LIN {X 0,Y 481.428,Z 376.763,A -85,B 0,C 180,E1 -7015.184,E2 -7015.184} C_VEL
LIN {X 0,Y 481.4,Z 381.681,A -85,B 0,C 180,E1 -7016.232,E2 -7016.232} C_VEL
LIN {X 0,Y 481.223,Z 384.559,A -85,B 0,C 180,E1 -7017.069,E2 -7017.069} C_VEL
LIN {X 0,Y 480.948,Z 387.393,A -85,B 0,C 180,E1 -7018.324,E2 -7018.324} C_VEL
LIN {X 0,Y 480.921,Z 388.409,A -85,B 0,C 180,E1 -7019.162,E2 -7019.162} C_VEL
LIN {X 0,Y 480.91,Z 388.742,A -85,B 0,C 180,E1 -7019.999,E2 -7019.999} C_VEL
LIN {X 0,Y 480.91,Z 388.397,A -85,B 0,C 180,E1 -7020.836,E2 -7020.836} C_VEL
LIN {X 0,Y 480.929,Z 387.368,A -85,B 0,C 180,E1 -7021.674,E2 -7021.674} C_VEL
LIN {X 0,Y 481.008,Z 385.622,A -85,B 0,C 180,E1 -7022.511,E2 -7022.511} C_VEL
LIN {X 0,Y 481.16,Z 383.117,A -85,B 0,C 180,E1 -7023.348,E2 -7023.348} C_VEL
LIN {X 0,Y 481.355,Z 379.786,A -85,B 0,C 180,E1 -7024.185,E2 -7024.185} C_VEL
LIN {X 0,Y 481.453,Z 374.316,A -85,B 0,C 180,E1 -7025.233,E2 -7025.233} C_VEL
LIN {X 0,Y 481.518,Z 368.474,A -85,B 0,C 180,E1 -7026.073,E2 -7026.073} C_VEL
LIN {X 0,Y 481.67,Z 361.279,A -85,B 0,C 180,E1 -7026.891,E2 -7026.891} C_VEL
LIN {X 0,Y 481.799,Z 353.733,A -85,B 0,C 180,E1 -7027.543,E2 -7027.543} C_VEL
LIN {X 0,Y 482.018,Z 344.137,A -85,B 0,C 180,E1 -7028.172,E2 -7028.172} C_VEL
LIN {X 0,Y 481.92,Z 337.555,A -85,B 0,C 180,E1 -7028.49,E2 -7028.49} C_VEL
LIN {X 0,Y 481.191,Z 332.773,A -85,B 0,C 180,E1 -7028.714,E2 -7028.714} C_VEL
LIN {X 0,Y 481.282,Z 325.199,A -85,B 0,C 180,E1 -7031.935,E2 -7031.935} C_VEL
LIN {X 0,Y 481.289,Z 316.966,A -85,B 0,C 180,E1 -7035.471,E2 -7035.471} C_VEL
LIN {X 0,Y 481.36,Z 309.359,A -85,B 0,C 180,E1 -7038.735,E2 -7038.735} C_VEL
LIN {X 0,Y 481.373,Z 303.142,A -85,B 0,C 180,E1 -7041.406,E2 -7041.406} C_VEL
LIN {X 0,Y 481.425,Z 296.779,A -85,B 0,C 180,E1 -7044.125,E2 -7044.125} C_VEL
LIN {X 0,Y 481.494,Z 289.818,A -85,B 0,C 180,E1 -7047.08,E2 -7047.08} C_VEL
LIN {X 0,Y 481.611,Z 284.497,A -85,B 0,C 180,E1 -7049.327,E2 -7049.327} C_VEL
LIN {X 0,Y 481.644,Z 284.486,A -85,B 0,C 180,E1 -7052.675,E2 -7052.675} C_VEL
LIN {X 0,Y 481.624,Z 284.489,A -85,B 0,C 180,E1 -7055.709,E2 -7055.709} C_VEL
LIN {X 0,Y 481.659,Z 284.49,A -85,B 0,C 180,E1 -7058.858,E2 -7058.858} C_VEL
LIN {X 0,Y 481.632,Z 284.489,A -85,B 0,C 180,E1 -7062.16,E2 -7062.16} C_VEL
LIN {X 0,Y 481.647,Z 284.486,A -85,B 0,C 180,E1 -7065.541,E2 -7065.541} C_VEL
LIN {X 0,Y 481.648,Z 284.488,A -85,B 0,C 180,E1 -7068.957,E2 -7068.957} C_VEL
LIN {X 0,Y 481.648,Z 284.49,A -85,B 0,C 180,E1 -7071.991,E2 -7071.991} C_VEL
LIN {X 0,Y 481.684,Z 284.483,A -85,B 0,C 180,E1 -7075.317,E2 -7075.317} C_VEL
LIN {X 0,Y 481.639,Z 284.49,A -85,B 0,C 180,E1 -7078.311,E2 -7078.311} C_VEL
LIN {X 0,Y 481.697,Z 284.484,A -85,B 0,C 180,E1 -7081.218,E2 -7081.218} C_VEL
LIN {X 0,Y 481.696,Z 284.483,A -85,B 0,C 180,E1 -7084.042,E2 -7084.042} C_VEL
LIN {X 0,Y 481.641,Z 284.488,A -85,B 0,C 180,E1 -7087.14,E2 -7087.14} C_VEL
LIN {X 0,Y 480.959,Z 284.576,A -85,B 0,C 180,E1 -7087.838,E2 -7087.838} C_VEL
LIN {X 0,Y 478.104,Z 284.933,A -85,B 0,C 180,E1 -7088.971,E2 -7088.971} C_VEL
LIN {X 0,Y 475.715,Z 285.227,A -85,B 0,C 180,E1 -7089.885,E2 -7089.885} C_VEL
LIN {X 0,Y 474.713,Z 285.353,A -85,B 0,C 180,E1 -7090.591,E2 -7090.591} C_VEL
LIN {X 0,Y 474.644,Z 285.362,A -85,B 0,C 180,E1 -7090.83,E2 -7090.83} C_VEL
LIN {X 0,Y 474.668,Z 285.357,A -85,B 0,C 180,E1 -7094.232,E2 -7094.232} C_VEL
LIN {X 0,Y 474.688,Z 285.353,A -85,B 0,C 180,E1 -7097.724,E2 -7097.724} C_VEL
LIN {X 0,Y 474.688,Z 285.357,A -85,B 0,C 180,E1 -7100.627,E2 -7100.627} C_VEL
LIN {X 0,Y 474.687,Z 285.353,A -85,B 0,C 180,E1 -7103.198,E2 -7103.198} C_VEL
LIN {X 0,Y 474.73,Z 285.348,A -85,B 0,C 180,E1 -7104.904,E2 -7104.904} C_VEL
LIN {X 0,Y 474.861,Z 285.331,A -85,B 0,C 180,E1 -7107.455,E2 -7107.455} C_VEL
LIN {X 0,Y 474.866,Z 285.337,A -85,B 0,C 180,E1 -7110,E2 -7110} C_VEL
LIN {X 0,Y 474.862,Z 285.331,A -85,B 0,C 180,E1 -7112.545,E2 -7112.545} C_VEL
LIN {X 0,Y 474.742,Z 285.35,A -85,B 0,C 180,E1 -7115.948,E2 -7115.948} C_VEL
LIN {X 0,Y 474.699,Z 285.352,A -85,B 0,C 180,E1 -7118.514,E2 -7118.514} C_VEL
LIN {X 0,Y 474.691,Z 285.354,A -85,B 0,C 180,E1 -7121.963,E2 -7121.963} C_VEL
LIN {X 0,Y 474.688,Z 285.357,A -85,B 0,C 180,E1 -7125.456,E2 -7125.456} C_VEL
LIN {X 0,Y 474.654,Z 285.362,A -85,B 0,C 180,E1 -7129.011,E2 -7129.011} C_VEL
LIN {X 0,Y 474.579,Z 285.368,A -85,B 0,C 180,E1 -7131.729,E2 -7131.729} C_VEL
LIN {X 0,Y 474.649,Z 285.362,A -85,B 0,C 180,E1 -7134.494,E2 -7134.494} C_VEL
LIN {X 0,Y 474.688,Z 285.354,A -85,B 0,C 180,E1 -7137.339,E2 -7137.339} C_VEL
LIN {X 0,Y 474.601,Z 285.366,A -85,B 0,C 180,E1 -7140.812,E2 -7140.812} C_VEL
LIN {X 0,Y 474.629,Z 285.365,A -85,B 0,C 180,E1 -7143.985,E2 -7143.985} C_VEL
LIN {X 0,Y 474.566,Z 285.369,A -85,B 0,C 180,E1 -7146.901,E2 -7146.901} C_VEL
LIN {X 0,Y 474.619,Z 285.366,A -85,B 0,C 180,E1 -7149.649,E2 -7149.649} C_VEL
LIN {X 0,Y 474.606,Z 285.365,A -85,B 0,C 180,E1 -7152.935,E2 -7152.935} C_VEL
LIN {X 0,Y 474.595,Z 285.366,A -85,B 0,C 180,E1 -7155.896,E2 -7155.896} C_VEL
LIN {X 0,Y 474.6,Z 285.37,A -85,B 0,C 180,E1 -7159.045,E2 -7159.045} C_VEL
LIN {X 0,Y 474.599,Z 285.364,A -85,B 0,C 180,E1 -7161.706,E2 -7161.706} C_VEL
LIN {X 0,Y 474.611,Z 285.368,A -85,B 0,C 180,E1 -7164.726,E2 -7164.726} C_VEL
LIN {X 0,Y 474.621,Z 285.36,A -85,B 0,C 180,E1 -7167.788,E2 -7167.788} C_VEL
LIN {X 0,Y 474.702,Z 285.409,A -85,B 0,C 180,E1 -7169.68,E2 -7169.68} C_VEL
LIN {X 0,Y 474.647,Z 289.554,A -85,B 0,C 180,E1 -7171.719,E2 -7171.719} C_VEL
LIN {X 0,Y 474.489,Z 295.509,A -85,B 0,C 180,E1 -7174.625,E2 -7174.625} C_VEL
LIN {X 0,Y 474.341,Z 301.144,A -85,B 0,C 180,E1 -7177.344,E2 -7177.344} C_VEL
LIN {X 0,Y 474.256,Z 306.861,A -85,B 0,C 180,E1 -7180.074,E2 -7180.074} C_VEL
LIN {X 0,Y 474.132,Z 312.578,A -85,B 0,C 180,E1 -7182.756,E2 -7182.756} C_VEL
LIN {X 0,Y 474.044,Z 318.251,A -85,B 0,C 180,E1 -7185.403,E2 -7185.403} C_VEL
LIN {X 0,Y 474.062,Z 324.061,A -85,B 0,C 180,E1 -7188.086,E2 -7188.086} C_VEL
LIN {X 0,Y 473.949,Z 330.434,A -85,B 0,C 180,E1 -7190.963,E2 -7190.963} C_VEL
LIN {X 0,Y 475.276,Z 340.728,A -85,B 0,C 180,E1 -7191.444,E2 -7191.444} C_VEL
LIN {X 0,Y 475.007,Z 350.2,A -85,B 0,C 180,E1 -7192.028,E2 -7192.028} C_VEL
LIN {X 0,Y 474.815,Z 358.727,A -85,B 0,C 180,E1 -7192.731,E2 -7192.731} C_VEL
LIN {X 0,Y 474.55,Z 367.023,A -85,B 0,C 180,E1 -7193.624,E2 -7193.624} C_VEL
LIN {X 0,Y 474.497,Z 373.154,A -85,B 0,C 180,E1 -7194.476,E2 -7194.476} C_VEL
LIN {X 0,Y 474.346,Z 379.082,A -85,B 0,C 180,E1 -7195.54,E2 -7195.54} C_VEL
LIN {X 0,Y 474.117,Z 383.478,A -85,B 0,C 180,E1 -7196.602,E2 -7196.602} C_VEL
LIN {X 0,Y 473.955,Z 386.076,A -85,B 0,C 180,E1 -7197.451,E2 -7197.451} C_VEL
LIN {X 0,Y 473.87,Z 387.921,A -85,B 0,C 180,E1 -7198.301,E2 -7198.301} C_VEL
LIN {X 0,Y 473.857,Z 389.063,A -85,B 0,C 180,E1 -7199.151,E2 -7199.151} C_VEL
LIN {X 0,Y 473.861,Z 389.533,A -85,B 0,C 180,E1 -7200.001,E2 -7200.001} C_VEL
LIN {X 0,Y 473.873,Z 389.335,A -85,B 0,C 180,E1 -7200.851,E2 -7200.851} C_VEL
LIN {X 0,Y 473.906,Z 388.472,A -85,B 0,C 180,E1 -7201.701,E2 -7201.701} C_VEL
LIN {X 0,Y 473.99,Z 386.922,A -85,B 0,C 180,E1 -7202.551,E2 -7202.551} C_VEL
LIN {X 0,Y 474.162,Z 384.636,A -85,B 0,C 180,E1 -7203.4,E2 -7203.4} C_VEL
LIN {X 0,Y 474.331,Z 381.561,A -85,B 0,C 180,E1 -7204.25,E2 -7204.25} C_VEL
LIN {X 0,Y 474.604,Z 376.463,A -85,B 0,C 180,E1 -7205.311,E2 -7205.311} C_VEL
LIN {X 0,Y 474.665,Z 371.191,A -85,B 0,C 180,E1 -7206.163,E2 -7206.163} C_VEL
LIN {X 0,Y 474.887,Z 364.006,A -85,B 0,C 180,E1 -7207.07,E2 -7207.07} C_VEL
LIN {X 0,Y 475.278,Z 354.988,A -85,B 0,C 180,E1 -7207.937,E2 -7207.937} C_VEL
LIN {X 0,Y 475.511,Z 345.724,A -85,B 0,C 180,E1 -7208.607,E2 -7208.607} C_VEL
LIN {X 0,Y 475.411,Z 339.085,A -85,B 0,C 180,E1 -7208.984,E2 -7208.984} C_VEL
LIN {X 0,Y 474.159,Z 332.143,A -85,B 0,C 180,E1 -7209.331,E2 -7209.331} C_VEL
LIN {X 0,Y 474.254,Z 326.504,A -85,B 0,C 180,E1 -7212.024,E2 -7212.024} C_VEL
LIN {X 0,Y 474.432,Z 319.008,A -85,B 0,C 180,E1 -7215.66,E2 -7215.66} C_VEL
LIN {X 0,Y 474.594,Z 312.239,A -85,B 0,C 180,E1 -7219.014,E2 -7219.014} C_VEL
LIN {X 0,Y 474.769,Z 306.861,A -85,B 0,C 180,E1 -7221.721,E2 -7221.721} C_VEL
LIN {X 0,Y 474.976,Z 301.509,A -85,B 0,C 180,E1 -7224.476,E2 -7224.476} C_VEL
LIN {X 0,Y 475.239,Z 295.854,A -85,B 0,C 180,E1 -7227.463,E2 -7227.463} C_VEL
LIN {X 0,Y 475.353,Z 290.917,A -85,B 0,C 180,E1 -7230.179,E2 -7230.179} C_VEL
LIN {X 0,Y 474.938,Z 286.999,A -85,B 0,C 180,E1 -7232.491,E2 -7232.491} C_VEL
LIN {X 0,Y 474.677,Z 285.361,A -85,B 0,C 180,E1 -7233.594,E2 -7233.594} C_VEL
LIN {X 0,Y 474.594,Z 285.37,A -85,B 0,C 180,E1 -7236.324,E2 -7236.324} C_VEL
LIN {X 0,Y 474.633,Z 285.365,A -85,B 0,C 180,E1 -7239.648,E2 -7239.648} C_VEL
LIN {X 0,Y 474.62,Z 285.367,A -85,B 0,C 180,E1 -7242.935,E2 -7242.935} C_VEL
LIN {X 0,Y 474.611,Z 285.367,A -85,B 0,C 180,E1 -7245.895,E2 -7245.895} C_VEL
LIN {X 0,Y 474.633,Z 285.366,A -85,B 0,C 180,E1 -7249.041,E2 -7249.041} C_VEL
LIN {X 0,Y 474.615,Z 285.368,A -85,B 0,C 180,E1 -7251.704,E2 -7251.704} C_VEL
LIN {X 0,Y 474.671,Z 285.497,A -85,B 0,C 180,E1 -7254.989,E2 -7254.989} C_VEL
LIN {X 0,Y 476.098,Z 291.334,A -85,B 0,C 180,E1 -7257.291,E2 -7257.291} C_VEL
LIN {X 0,Y 477.894,Z 299.615,A -85,B 0,C 180,E1 -7259.999,E2 -7259.999} C_VEL
LIN {X 0,Y 478.476,Z 303.1,A -85,B 0,C 180,E1 -7261.006,E2 -7261.006} C_VEL
LIN {X 0,Y 478.091,Z 308.638,A -85,B 0,C 180,E1 -7262.415,E2 -7262.415} C_VEL
LIN {X 0,Y 476.789,Z 322.51,A -85,B 0,C 180,E1 -7265.624,E2 -7265.624} C_VEL
LIN {X 0,Y 475.729,Z 339.255,A -85,B 0,C 180,E1 -7269.234,E2 -7269.234} C_VEL
LIN {X 0,Y 475.019,Z 355.708,A -85,B 0,C 180,E1 -7272.566,E2 -7272.566} C_VEL
LIN {X 0,Y 474.627,Z 369.075,A -85,B 0,C 180,E1 -7275.174,E2 -7275.174} C_VEL
LIN {X 0,Y 476.028,Z 383.097,A -85,B 0,C 180,E1 -7275.546,E2 -7275.546} C_VEL
LIN {X 0,Y 476.321,Z 388.808,A -85,B 0,C 180,E1 -7275.746,E2 -7275.746} C_VEL
LIN {X 0,Y 475.977,Z 401.249,A -85,B 0,C 180,E1 -7276.28,E2 -7276.28} C_VEL
LIN {X 0,Y 475.522,Z 413.187,A -85,B 0,C 180,E1 -7276.974,E2 -7276.974} C_VEL
LIN {X 0,Y 475.283,Z 423.595,A -85,B 0,C 180,E1 -7277.746,E2 -7277.746} C_VEL
LIN {X 0,Y 474.806,Z 433.942,A -85,B 0,C 180,E1 -7278.69,E2 -7278.69} C_VEL
LIN {X 0,Y 474.46,Z 443.425,A -85,B 0,C 180,E1 -7279.761,E2 -7279.761} C_VEL
LIN {X 0,Y 474.221,Z 452.603,A -85,B 0,C 180,E1 -7281.048,E2 -7281.048} C_VEL
LIN {X 0,Y 474.043,Z 459.976,A -85,B 0,C 180,E1 -7282.332,E2 -7282.332} C_VEL
LIN {X 0,Y 473.877,Z 466.576,A -85,B 0,C 180,E1 -7283.809,E2 -7283.809} C_VEL
LIN {X 0,Y 473.852,Z 470.404,A -85,B 0,C 180,E1 -7284.894,E2 -7284.894} C_VEL
LIN {X 0,Y 473.898,Z 472.829,A -85,B 0,C 180,E1 -7285.748,E2 -7285.748} C_VEL
LIN {X 0,Y 473.92,Z 474.806,A -85,B 0,C 180,E1 -7286.599,E2 -7286.599} C_VEL
LIN {X 0,Y 473.883,Z 476.298,A -85,B 0,C 180,E1 -7287.45,E2 -7287.45} C_VEL
LIN {X 0,Y 473.758,Z 478.001,A -85,B 0,C 180,E1 -7289.15,E2 -7289.15} C_VEL
LIN {X 0,Y 473.761,Z 478.249,A -85,B 0,C 180,E1 -7290,E2 -7290} C_VEL
LIN {X 0,Y 473.754,Z 478.042,A -85,B 0,C 180,E1 -7290.85,E2 -7290.85} C_VEL
LIN {X 0,Y 473.881,Z 476.432,A -85,B 0,C 180,E1 -7292.55,E2 -7292.55} C_VEL
LIN {X 0,Y 473.904,Z 474.976,A -85,B 0,C 180,E1 -7293.401,E2 -7293.401} C_VEL
LIN {X 0,Y 473.81,Z 471.936,A -85,B 0,C 180,E1 -7294.679,E2 -7294.679} C_VEL
LIN {X 0,Y 473.905,Z 467.814,A -85,B 0,C 180,E1 -7295.959,E2 -7295.959} C_VEL
LIN {X 0,Y 474.017,Z 461.448,A -85,B 0,C 180,E1 -7297.454,E2 -7297.454} C_VEL
LIN {X 0,Y 474.181,Z 454.486,A -85,B 0,C 180,E1 -7298.738,E2 -7298.738} C_VEL
LIN {X 0,Y 474.428,Z 445.714,A -85,B 0,C 180,E1 -7300.024,E2 -7300.024} C_VEL
LIN {X 0,Y 474.835,Z 435.719,A -85,B 0,C 180,E1 -7301.202,E2 -7301.202} C_VEL
LIN {X 0,Y 475.243,Z 426.23,A -85,B 0,C 180,E1 -7302.105,E2 -7302.105} C_VEL
LIN {X 0,Y 475.538,Z 415.711,A -85,B 0,C 180,E1 -7302.917,E2 -7302.917} C_VEL
LIN {X 0,Y 475.936,Z 403.316,A -85,B 0,C 180,E1 -7303.666,E2 -7303.666} C_VEL
LIN {X 0,Y 476.298,Z 391.532,A -85,B 0,C 180,E1 -7304.2,E2 -7304.2} C_VEL
LIN {X 0,Y 476.195,Z 383.965,A -85,B 0,C 180,E1 -7304.462,E2 -7304.462} C_VEL
LIN {X 0,Y 474.685,Z 369.599,A -85,B 0,C 180,E1 -7304.852,E2 -7304.852} C_VEL
LIN {X 0,Y 475.239,Z 353.202,A -85,B 0,C 180,E1 -7308.093,E2 -7308.093} C_VEL
LIN {X 0,Y 476.031,Z 335.475,A -85,B 0,C 180,E1 -7311.66,E2 -7311.66} C_VEL
LIN {X 0,Y 476.93,Z 318.979,A -85,B 0,C 180,E1 -7315.066,E2 -7315.066} C_VEL
LIN {X 0,Y 477.984,Z 303.66,A -85,B 0,C 180,E1 -7318.306,E2 -7318.306} C_VEL
LIN {X 0,Y 477.87,Z 300.392,A -85,B 0,C 180,E1 -7319.034,E2 -7319.034} C_VEL
LIN {X 0,Y 475.231,Z 288.352,A -85,B 0,C 180,E1 -7321.917,E2 -7321.917} C_VEL
LIN {X 0,Y 474.647,Z 285.363,A -85,B 0,C 180,E1 -7322.677,E2 -7322.677} C_VEL
LIN {X 0,Y 474.618,Z 285.367,A -85,B 0,C 180,E1 -7325.469,E2 -7325.469} C_VEL
LIN {X 0,Y 474.617,Z 285.368,A -85,B 0,C 180,E1 -7328.457,E2 -7328.457} C_VEL
LIN {X 0,Y 474.633,Z 285.364,A -85,B 0,C 180,E1 -7330.959,E2 -7330.959} C_VEL
LIN {X 0,Y 474.615,Z 285.367,A -85,B 0,C 180,E1 -7334.105,E2 -7334.105} C_VEL
LIN {X 0,Y 474.62,Z 285.366,A -85,B 0,C 180,E1 -7337.065,E2 -7337.065} C_VEL
LIN {X 0,Y 474.65,Z 285.363,A -85,B 0,C 180,E1 -7340.454,E2 -7340.454} C_VEL
LIN {X 0,Y 474.594,Z 285.37,A -85,B 0,C 180,E1 -7343.676,E2 -7343.676} C_VEL
LIN {X 0,Y 474.63,Z 285.368,A -85,B 0,C 180,E1 -7346.778,E2 -7346.778} C_VEL
LIN {X 0,Y 474.552,Z 285.377,A -85,B 0,C 180,E1 -7349.765,E2 -7349.765} C_VEL
LIN {X 0,Y 474.472,Z 285.527,A -85,B 0,C 180,E1 -7351.585,E2 -7351.585} C_VEL
LIN {X 0,Y 474.439,Z 293.989,A -85,B 0,C 180,E1 -7354.637,E2 -7354.637} C_VEL
LIN {X 0,Y 474.425,Z 302.282,A -85,B 0,C 180,E1 -7357.805,E2 -7357.805} C_VEL
LIN {X 0,Y 474.405,Z 308.984,A -85,B 0,C 180,E1 -7360.528,E2 -7360.528} C_VEL
LIN {X 0,Y 474.364,Z 315.627,A -85,B 0,C 180,E1 -7363.207,E2 -7363.207} C_VEL
LIN {X 0,Y 474.329,Z 321.965,A -85,B 0,C 180,E1 -7365.848,E2 -7365.848} C_VEL
LIN {X 0,Y 474.35,Z 328.129,A -85,B 0,C 180,E1 -7368.461,E2 -7368.461} C_VEL
LIN {X 0,Y 474.349,Z 334.862,A -85,B 0,C 180,E1 -7371.251,E2 -7371.251} C_VEL
LIN {X 0,Y 475.167,Z 341.473,A -85,B 0,C 180,E1 -7371.547,E2 -7371.547} C_VEL
LIN {X 0,Y 475.004,Z 349.921,A -85,B 0,C 180,E1 -7372.026,E2 -7372.026} C_VEL
LIN {X 0,Y 474.874,Z 358.028,A -85,B 0,C 180,E1 -7372.634,E2 -7372.634} C_VEL
LIN {X 0,Y 474.532,Z 365.791,A -85,B 0,C 180,E1 -7373.408,E2 -7373.408} C_VEL
LIN {X 0,Y 474.592,Z 372.407,A -85,B 0,C 180,E1 -7374.262,E2 -7374.262} C_VEL
LIN {X 0,Y 474.402,Z 377.489,A -85,B 0,C 180,E1 -7375.112,E2 -7375.112} C_VEL
LIN {X 0,Y 474.371,Z 382.385,A -85,B 0,C 180,E1 -7376.176,E2 -7376.176} C_VEL
LIN {X 0,Y 474.182,Z 385.253,A -85,B 0,C 180,E1 -7377.025,E2 -7377.025} C_VEL
LIN {X 0,Y 473.885,Z 388.074,A -85,B 0,C 180,E1 -7378.299,E2 -7378.299} C_VEL
LIN {X 0,Y 473.854,Z 389.083,A -85,B 0,C 180,E1 -7379.149,E2 -7379.149} C_VEL
LIN {X 0,Y 473.842,Z 389.406,A -85,B 0,C 180,E1 -7379.999,E2 -7379.999} C_VEL
LIN {X 0,Y 473.842,Z 389.048,A -85,B 0,C 180,E1 -7380.849,E2 -7380.849} C_VEL
LIN {X 0,Y 473.862,Z 388.004,A -85,B 0,C 180,E1 -7381.699,E2 -7381.699} C_VEL
LIN {X 0,Y 473.952,Z 386.24,A -85,B 0,C 180,E1 -7382.549,E2 -7382.549} C_VEL
LIN {X 0,Y 474.116,Z 383.714,A -85,B 0,C 180,E1 -7383.398,E2 -7383.398} C_VEL
LIN {X 0,Y 474.325,Z 380.358,A -85,B 0,C 180,E1 -7384.247,E2 -7384.247} C_VEL
LIN {X 0,Y 474.419,Z 374.853,A -85,B 0,C 180,E1 -7385.311,E2 -7385.311} C_VEL
LIN {X 0,Y 474.495,Z 368.977,A -85,B 0,C 180,E1 -7386.163,E2 -7386.163} C_VEL
LIN {X 0,Y 474.638,Z 361.739,A -85,B 0,C 180,E1 -7386.993,E2 -7386.993} C_VEL
LIN {X 0,Y 474.774,Z 354.145,A -85,B 0,C 180,E1 -7387.655,E2 -7387.655} C_VEL
LIN {X 0,Y 474.998,Z 346.335,A -85,B 0,C 180,E1 -7388.186,E2 -7388.186} C_VEL
LIN {X 0,Y 474.821,Z 337.786,A -85,B 0,C 180,E1 -7388.618,E2 -7388.618} C_VEL
LIN {X 0,Y 474.166,Z 333.348,A -85,B 0,C 180,E1 -7388.818,E2 -7388.818} C_VEL
LIN {X 0,Y 474.242,Z 325.829,A -85,B 0,C 180,E1 -7392.017,E2 -7392.017} C_VEL
LIN {X 0,Y 474.232,Z 317.553,A -85,B 0,C 180,E1 -7395.573,E2 -7395.573} C_VEL
LIN {X 0,Y 474.325,Z 309.54,A -85,B 0,C 180,E1 -7399.023,E2 -7399.023} C_VEL
LIN {X 0,Y 474.339,Z 303.215,A -85,B 0,C 180,E1 -7401.739,E2 -7401.739} C_VEL
LIN {X 0,Y 474.396,Z 295.785,A -85,B 0,C 180,E1 -7404.928,E2 -7404.928} C_VEL
LIN {X 0,Y 474.509,Z 287.825,A -85,B 0,C 180,E1 -7408.29,E2 -7408.29} C_VEL
LIN {X 0,Y 474.587,Z 285.372,A -85,B 0,C 180,E1 -7409.374,E2 -7409.374} C_VEL
LIN {X 0,Y 474.591,Z 285.364,A -85,B 0,C 180,E1 -7412.425,E2 -7412.425} C_VEL
LIN {X 0,Y 474.603,Z 285.366,A -85,B 0,C 180,E1 -7415.467,E2 -7415.467} C_VEL
LIN {X 0,Y 474.601,Z 285.365,A -85,B 0,C 180,E1 -7418.456,E2 -7418.456} C_VEL
LIN {X 0,Y 474.601,Z 285.364,A -85,B 0,C 180,E1 -7421.785,E2 -7421.785} C_VEL
LIN {X 0,Y 474.608,Z 285.369,A -85,B 0,C 180,E1 -7424.701,E2 -7424.701} C_VEL
LIN {X 0,Y 474.617,Z 285.363,A -85,B 0,C 180,E1 -7427.762,E2 -7427.762} C_VEL
LIN {X 0,Y 474.636,Z 285.365,A -85,B 0,C 180,E1 -7430.453,E2 -7430.453} C_VEL
LIN {X 0,Y 474.585,Z 285.37,A -85,B 0,C 180,E1 -7433.676,E2 -7433.676} C_VEL
LIN {X 0,Y 474.634,Z 285.361,A -85,B 0,C 180,E1 -7436.779,E2 -7436.779} C_VEL
LIN {X 0,Y 474.604,Z 285.367,A -85,B 0,C 180,E1 -7439.77,E2 -7439.77} C_VEL
LIN {X 0,Y 474.704,Z 285.352,A -85,B 0,C 180,E1 -7442.68,E2 -7442.68} C_VEL
LIN {X 0,Y 474.649,Z 285.362,A -85,B 0,C 180,E1 -7445.506,E2 -7445.506} C_VEL
LIN {X 0,Y 474.659,Z 285.361,A -85,B 0,C 180,E1 -7449.185,E2 -7449.185} C_VEL
LIN {X 0,Y 474.644,Z 285.362,A -85,B 0,C 180,E1 -7450.83,E2 -7450.83} C_VEL
LIN {X 0,Y 474.014,Z 285.445,A -85,B 0,C 180,E1 -7451.538,E2 -7451.538} C_VEL
LIN {X 0,Y 471.186,Z 285.798,A -85,B 0,C 180,E1 -7452.688,E2 -7452.688} C_VEL
LIN {X 0,Y 468.761,Z 286.096,A -85,B 0,C 180,E1 -7453.615,E2 -7453.615} C_VEL
LIN {X 0,Y 467.7,Z 286.226,A -85,B 0,C 180,E1 -7454.331,E2 -7454.331} C_VEL
LIN {X 0,Y 467.605,Z 286.236,A -85,B 0,C 180,E1 -7454.574,E2 -7454.574} C_VEL
LIN {X 0,Y 467.643,Z 286.231,A -85,B 0,C 180,E1 -7457.854,E2 -7457.854} C_VEL
LIN {X 0,Y 467.657,Z 286.229,A -85,B 0,C 180,E1 -7461.357,E2 -7461.357} C_VEL
LIN {X 0,Y 467.704,Z 286.226,A -85,B 0,C 180,E1 -7463.962,E2 -7463.962} C_VEL
LIN {X 0,Y 467.802,Z 286.21,A -85,B 0,C 180,E1 -7467.417,E2 -7467.417} C_VEL
LIN {X 0,Y 467.836,Z 286.213,A -85,B 0,C 180,E1 -7470,E2 -7470} C_VEL
LIN {X 0,Y 467.802,Z 286.21,A -85,B 0,C 180,E1 -7472.583,E2 -7472.583} C_VEL
LIN {X 0,Y 467.705,Z 286.226,A -85,B 0,C 180,E1 -7476.038,E2 -7476.038} C_VEL
LIN {X 0,Y 467.657,Z 286.229,A -85,B 0,C 180,E1 -7478.643,E2 -7478.643} C_VEL
LIN {X 0,Y 467.643,Z 286.231,A -85,B 0,C 180,E1 -7482.146,E2 -7482.146} C_VEL
LIN {X 0,Y 467.627,Z 286.235,A -85,B 0,C 180,E1 -7485.695,E2 -7485.695} C_VEL
LIN {X 0,Y 467.606,Z 286.239,A -85,B 0,C 180,E1 -7488.765,E2 -7488.765} C_VEL
LIN {X 0,Y 467.57,Z 286.243,A -85,B 0,C 180,E1 -7491.269,E2 -7491.269} C_VEL
LIN {X 0,Y 467.562,Z 286.243,A -85,B 0,C 180,E1 -7493.944,E2 -7493.944} C_VEL
LIN {X 0,Y 467.618,Z 286.239,A -85,B 0,C 180,E1 -7496.8,E2 -7496.8} C_VEL
LIN {X 0,Y 467.578,Z 286.242,A -85,B 0,C 180,E1 -7499.737,E2 -7499.737} C_VEL
LIN {X 0,Y 467.574,Z 286.241,A -85,B 0,C 180,E1 -7502.759,E2 -7502.759} C_VEL
LIN {X 0,Y 467.548,Z 286.247,A -85,B 0,C 180,E1 -7505.89,E2 -7505.89} C_VEL
LIN {X 0,Y 467.574,Z 286.242,A -85,B 0,C 180,E1 -7509.146,E2 -7509.146} C_VEL
LIN {X 0,Y 467.579,Z 286.239,A -85,B 0,C 180,E1 -7512.568,E2 -7512.568} C_VEL
LIN {X 0,Y 467.558,Z 286.245,A -85,B 0,C 180,E1 -7515.054,E2 -7515.054} C_VEL
LIN {X 0,Y 467.559,Z 286.242,A -85,B 0,C 180,E1 -7518.597,E2 -7518.597} C_VEL
LIN {X 0,Y 467.554,Z 286.241,A -85,B 0,C 180,E1 -7521.956,E2 -7521.956} C_VEL
LIN {X 0,Y 467.548,Z 286.244,A -85,B 0,C 180,E1 -7525.168,E2 -7525.168} C_VEL
LIN {X 0,Y 467.583,Z 286.24,A -85,B 0,C 180,E1 -7528.262,E2 -7528.262} C_VEL
LIN {X 0,Y 467.658,Z 286.322,A -85,B 0,C 180,E1 -7529.649,E2 -7529.649} C_VEL
LIN {X 0,Y 467.604,Z 291.992,A -85,B 0,C 180,E1 -7532.469,E2 -7532.469} C_VEL
LIN {X 0,Y 467.395,Z 297.385,A -85,B 0,C 180,E1 -7535.102,E2 -7535.102} C_VEL
LIN {X 0,Y 467.262,Z 303.164,A -85,B 0,C 180,E1 -7537.914,E2 -7537.914} C_VEL
LIN {X 0,Y 467.185,Z 308.921,A -85,B 0,C 180,E1 -7540.675,E2 -7540.675} C_VEL
LIN {X 0,Y 467.032,Z 314.647,A -85,B 0,C 180,E1 -7543.388,E2 -7543.388} C_VEL
LIN {X 0,Y 466.937,Z 320.368,A -85,B 0,C 180,E1 -7546.066,E2 -7546.066} C_VEL
LIN {X 0,Y 466.93,Z 326.096,A -85,B 0,C 180,E1 -7548.717,E2 -7548.717} C_VEL
LIN {X 0,Y 466.88,Z 330.638,A -85,B 0,C 180,E1 -7550.798,E2 -7550.798} C_VEL
LIN {X 0,Y 468.307,Z 341.362,A -85,B 0,C 180,E1 -7551.316,E2 -7551.316} C_VEL
LIN {X 0,Y 468,Z 350.754,A -85,B 0,C 180,E1 -7551.908,E2 -7551.908} C_VEL
LIN {X 0,Y 467.792,Z 359.558,A -85,B 0,C 180,E1 -7552.65,E2 -7552.65} C_VEL
LIN {X 0,Y 467.534,Z 367.548,A -85,B 0,C 180,E1 -7553.528,E2 -7553.528} C_VEL
LIN {X 0,Y 467.462,Z 373.695,A -85,B 0,C 180,E1 -7554.393,E2 -7554.393} C_VEL
LIN {X 0,Y 467.318,Z 379.644,A -85,B 0,C 180,E1 -7555.473,E2 -7555.473} C_VEL
LIN {X 0,Y 467.075,Z 384.063,A -85,B 0,C 180,E1 -7556.551,E2 -7556.551} C_VEL
LIN {X 0,Y 466.901,Z 386.685,A -85,B 0,C 180,E1 -7557.413,E2 -7557.413} C_VEL
LIN {X 0,Y 466.803,Z 388.555,A -85,B 0,C 180,E1 -7558.276,E2 -7558.276} C_VEL
LIN {X 0,Y 466.79,Z 389.721,A -85,B 0,C 180,E1 -7559.138,E2 -7559.138} C_VEL
LIN {X 0,Y 466.795,Z 390.215,A -85,B 0,C 180,E1 -7560.001,E2 -7560.001} C_VEL
LIN {X 0,Y 466.81,Z 390.042,A -85,B 0,C 180,E1 -7560.864,E2 -7560.864} C_VEL
LIN {X 0,Y 466.847,Z 389.203,A -85,B 0,C 180,E1 -7561.726,E2 -7561.726} C_VEL
LIN {X 0,Y 466.938,Z 387.677,A -85,B 0,C 180,E1 -7562.589,E2 -7562.589} C_VEL
LIN {X 0,Y 467.123,Z 385.417,A -85,B 0,C 180,E1 -7563.451,E2 -7563.451} C_VEL
LIN {X 0,Y 467.304,Z 382.367,A -85,B 0,C 180,E1 -7564.314,E2 -7564.314} C_VEL
LIN {X 0,Y 467.592,Z 377.315,A -85,B 0,C 180,E1 -7565.391,E2 -7565.391} C_VEL
LIN {X 0,Y 467.667,Z 372.082,A -85,B 0,C 180,E1 -7566.256,E2 -7566.256} C_VEL
LIN {X 0,Y 467.911,Z 365.095,A -85,B 0,C 180,E1 -7567.163,E2 -7567.163} C_VEL
LIN {X 0,Y 468.284,Z 357.189,A -85,B 0,C 180,E1 -7567.959,E2 -7567.959} C_VEL
LIN {X 0,Y 468.517,Z 348.659,A -85,B 0,C 180,E1 -7568.628,E2 -7568.628} C_VEL
LIN {X 0,Y 468.681,Z 341.662,A -85,B 0,C 180,E1 -7569.06,E2 -7569.06} C_VEL
LIN {X 0,Y 467.092,Z 332.581,A -85,B 0,C 180,E1 -7569.555,E2 -7569.555} C_VEL
LIN {X 0,Y 467.227,Z 327.184,A -85,B 0,C 180,E1 -7572.158,E2 -7572.158} C_VEL
LIN {X 0,Y 467.418,Z 319.823,A -85,B 0,C 180,E1 -7575.784,E2 -7575.784} C_VEL
LIN {X 0,Y 467.604,Z 313.927,A -85,B 0,C 180,E1 -7578.759,E2 -7578.759} C_VEL
LIN {X 0,Y 467.783,Z 307.416,A -85,B 0,C 180,E1 -7582.062,E2 -7582.062} C_VEL
LIN {X 0,Y 468.043,Z 302.109,A -85,B 0,C 180,E1 -7584.863,E2 -7584.863} C_VEL
LIN {X 0,Y 468.316,Z 296.863,A -85,B 0,C 180,E1 -7587.725,E2 -7587.725} C_VEL
LIN {X 0,Y 468.456,Z 293.391,A -85,B 0,C 180,E1 -7589.676,E2 -7589.676} C_VEL
LIN {X 0,Y 468.204,Z 290.024,A -85,B 0,C 180,E1 -7591.694,E2 -7591.694} C_VEL
LIN {X 0,Y 467.594,Z 286.244,A -85,B 0,C 180,E1 -7594.243,E2 -7594.243} C_VEL
LIN {X 0,Y 467.553,Z 286.247,A -85,B 0,C 180,E1 -7597.187,E2 -7597.187} C_VEL
LIN {X 0,Y 467.583,Z 286.243,A -85,B 0,C 180,E1 -7600.265,E2 -7600.265} C_VEL
LIN {X 0,Y 467.592,Z 286.243,A -85,B 0,C 180,E1 -7602.567,E2 -7602.567} C_VEL
LIN {X 0,Y 467.571,Z 286.244,A -85,B 0,C 180,E1 -7605.053,E2 -7605.053} C_VEL
LIN {X 0,Y 467.594,Z 286.242,A -85,B 0,C 180,E1 -7607.44,E2 -7607.44} C_VEL
LIN {X 0,Y 467.587,Z 286.243,A -85,B 0,C 180,E1 -7610.856,E2 -7610.856} C_VEL
LIN {X 0,Y 467.576,Z 286.316,A -85,B 0,C 180,E1 -7614.168,E2 -7614.168} C_VEL
LIN {X 0,Y 468.787,Z 291.196,A -85,B 0,C 180,E1 -7616.31,E2 -7616.31} C_VEL
LIN {X 0,Y 470.127,Z 297.038,A -85,B 0,C 180,E1 -7618.451,E2 -7618.451} C_VEL
LIN {X 0,Y 471.518,Z 303.628,A -85,B 0,C 180,E1 -7620.537,E2 -7620.537} C_VEL
LIN {X 0,Y 471.596,Z 307.295,A -85,B 0,C 180,E1 -7621.554,E2 -7621.554} C_VEL
LIN {X 0,Y 470.297,Z 318.611,A -85,B 0,C 180,E1 -7624.318,E2 -7624.318} C_VEL
LIN {X 0,Y 469.201,Z 331.78,A -85,B 0,C 180,E1 -7627.313,E2 -7627.313} C_VEL
LIN {X 0,Y 468.602,Z 342.338,A -85,B 0,C 180,E1 -7629.592,E2 -7629.592} C_VEL
LIN {X 0,Y 467.983,Z 356.527,A -85,B 0,C 180,E1 -7632.521,E2 -7632.521} C_VEL
LIN {X 0,Y 467.585,Z 368.934,A -85,B 0,C 180,E1 -7634.973,E2 -7634.973} C_VEL
LIN {X 0,Y 468.913,Z 382.282,A -85,B 0,C 180,E1 -7635.336,E2 -7635.336} C_VEL
LIN {X 0,Y 469.345,Z 389.149,A -85,B 0,C 180,E1 -7635.585,E2 -7635.585} C_VEL
LIN {X 0,Y 469.018,Z 401.322,A -85,B 0,C 180,E1 -7636.128,E2 -7636.128} C_VEL
LIN {X 0,Y 468.505,Z 413.88,A -85,B 0,C 180,E1 -7636.886,E2 -7636.886} C_VEL
LIN {X 0,Y 468.217,Z 424.881,A -85,B 0,C 180,E1 -7637.739,E2 -7637.739} C_VEL
LIN {X 0,Y 467.746,Z 435.17,A -85,B 0,C 180,E1 -7638.736,E2 -7638.736} C_VEL
LIN {X 0,Y 467.367,Z 444.307,A -85,B 0,C 180,E1 -7639.823,E2 -7639.823} C_VEL
LIN {X 0,Y 467.108,Z 453.216,A -85,B 0,C 180,E1 -7641.128,E2 -7641.128} C_VEL
LIN {X 0,Y 466.95,Z 460.295,A -85,B 0,C 180,E1 -7642.432,E2 -7642.432} C_VEL
LIN {X 0,Y 466.805,Z 466.777,A -85,B 0,C 180,E1 -7643.95,E2 -7643.95} C_VEL
LIN {X 0,Y 466.744,Z 470.999,A -85,B 0,C 180,E1 -7645.25,E2 -7645.25} C_VEL
LIN {X 0,Y 466.845,Z 474.129,A -85,B 0,C 180,E1 -7646.548,E2 -7646.548} C_VEL
LIN {X 0,Y 466.826,Z 475.632,A -85,B 0,C 180,E1 -7647.411,E2 -7647.411} C_VEL
LIN {X 0,Y 466.687,Z 477.344,A -85,B 0,C 180,E1 -7649.137,E2 -7649.137} C_VEL
LIN {X 0,Y 466.691,Z 477.593,A -85,B 0,C 180,E1 -7650,E2 -7650} C_VEL
LIN {X 0,Y 466.684,Z 477.386,A -85,B 0,C 180,E1 -7650.863,E2 -7650.863} C_VEL
LIN {X 0,Y 466.824,Z 475.775,A -85,B 0,C 180,E1 -7652.589,E2 -7652.589} C_VEL
LIN {X 0,Y 466.829,Z 474.307,A -85,B 0,C 180,E1 -7653.452,E2 -7653.452} C_VEL
LIN {X 0,Y 466.732,Z 471.254,A -85,B 0,C 180,E1 -7654.751,E2 -7654.751} C_VEL
LIN {X 0,Y 466.804,Z 467.112,A -85,B 0,C 180,E1 -7656.05,E2 -7656.05} C_VEL
LIN {X 0,Y 466.94,Z 461.748,A -85,B 0,C 180,E1 -7657.35,E2 -7657.35} C_VEL
LIN {X 0,Y 467.102,Z 454.984,A -85,B 0,C 180,E1 -7658.654,E2 -7658.654} C_VEL
LIN {X 0,Y 467.307,Z 446.542,A -85,B 0,C 180,E1 -7659.96,E2 -7659.96} C_VEL
LIN {X 0,Y 467.688,Z 437.81,A -85,B 0,C 180,E1 -7661.046,E2 -7661.046} C_VEL
LIN {X 0,Y 468.102,Z 428.202,A -85,B 0,C 180,E1 -7662.024,E2 -7662.024} C_VEL
LIN {X 0,Y 468.449,Z 417.233,A -85,B 0,C 180,E1 -7662.929,E2 -7662.929} C_VEL
LIN {X 0,Y 468.869,Z 406.027,A -85,B 0,C 180,E1 -7663.655,E2 -7663.655} C_VEL
LIN {X 0,Y 469.259,Z 393.924,A -85,B 0,C 180,E1 -7664.252,E2 -7664.252} C_VEL
LIN {X 0,Y 469.275,Z 385.197,A -85,B 0,C 180,E1 -7664.583,E2 -7664.583} C_VEL
LIN {X 0,Y 467.889,Z 371.759,A -85,B 0,C 180,E1 -7664.961,E2 -7664.961} C_VEL
LIN {X 0,Y 467.618,Z 369.362,A -85,B 0,C 180,E1 -7665.026,E2 -7665.026} C_VEL
LIN {X 0,Y 468.187,Z 353.869,A -85,B 0,C 180,E1 -7668.149,E2 -7668.149} C_VEL
LIN {X 0,Y 469.022,Z 336.513,A -85,B 0,C 180,E1 -7671.714,E2 -7671.714} C_VEL
LIN {X 0,Y 469.916,Z 320.901,A -85,B 0,C 180,E1 -7674.993,E2 -7674.993} C_VEL
LIN {X 0,Y 471.038,Z 305.438,A -85,B 0,C 180,E1 -7678.321,E2 -7678.321} C_VEL
LIN {X 0,Y 471.039,Z 302.385,A -85,B 0,C 180,E1 -7679.006,E2 -7679.006} C_VEL
LIN {X 0,Y 468.676,Z 291.435,A -85,B 0,C 180,E1 -7681.658,E2 -7681.658} C_VEL
LIN {X 0,Y 467.592,Z 286.243,A -85,B 0,C 180,E1 -7683.014,E2 -7683.014} C_VEL
LIN {X 0,Y 467.558,Z 286.246,A -85,B 0,C 180,E1 -7685.889,E2 -7685.889} C_VEL
LIN {X 0,Y 467.587,Z 286.242,A -85,B 0,C 180,E1 -7689.144,E2 -7689.144} C_VEL
LIN {X 0,Y 467.592,Z 286.243,A -85,B 0,C 180,E1 -7692.567,E2 -7692.567} C_VEL
LIN {X 0,Y 467.576,Z 286.243,A -85,B 0,C 180,E1 -7695.053,E2 -7695.053} C_VEL
LIN {X 0,Y 467.594,Z 286.241,A -85,B 0,C 180,E1 -7697.44,E2 -7697.44} C_VEL
LIN {X 0,Y 467.588,Z 286.242,A -85,B 0,C 180,E1 -7700.855,E2 -7700.855} C_VEL
LIN {X 0,Y 467.564,Z 286.246,A -85,B 0,C 180,E1 -7704.261,E2 -7704.261} C_VEL
LIN {X 0,Y 467.585,Z 286.246,A -85,B 0,C 180,E1 -7707.321,E2 -7707.321} C_VEL
LIN {X 0,Y 467.491,Z 286.255,A -85,B 0,C 180,E1 -7710.257,E2 -7710.257} C_VEL
LIN {X 0,Y 467.457,Z 286.337,A -85,B 0,C 180,E1 -7711.426,E2 -7711.426} C_VEL
LIN {X 0,Y 467.456,Z 294.603,A -85,B 0,C 180,E1 -7714.433,E2 -7714.433} C_VEL
LIN {X 0,Y 467.407,Z 302.511,A -85,B 0,C 180,E1 -7717.453,E2 -7717.453} C_VEL
LIN {X 0,Y 467.413,Z 309.438,A -85,B 0,C 180,E1 -7720.225,E2 -7720.225} C_VEL
LIN {X 0,Y 467.332,Z 317.087,A -85,B 0,C 180,E1 -7723.396,E2 -7723.396} C_VEL
LIN {X 0,Y 467.335,Z 322.532,A -85,B 0,C 180,E1 -7725.632,E2 -7725.632} C_VEL
LIN {X 0,Y 467.338,Z 329.815,A -85,B 0,C 180,E1 -7728.725,E2 -7728.725} C_VEL
LIN {X 0,Y 467.311,Z 335.326,A -85,B 0,C 180,E1 -7731.077,E2 -7731.077} C_VEL
LIN {X 0,Y 468.211,Z 341.388,A -85,B 0,C 180,E1 -7731.366,E2 -7731.366} C_VEL
LIN {X 0,Y 468.015,Z 350.845,A -85,B 0,C 180,E1 -7731.906,E2 -7731.906} C_VEL
LIN {X 0,Y 467.879,Z 359.152,A -85,B 0,C 180,E1 -7732.547,E2 -7732.547} C_VEL
LIN {X 0,Y 467.545,Z 366.617,A -85,B 0,C 180,E1 -7733.309,E2 -7733.309} C_VEL
LIN {X 0,Y 467.576,Z 373.203,A -85,B 0,C 180,E1 -7734.176,E2 -7734.176} C_VEL
LIN {X 0,Y 467.377,Z 378.265,A -85,B 0,C 180,E1 -7735.039,E2 -7735.039} C_VEL
LIN {X 0,Y 467.342,Z 383.142,A -85,B 0,C 180,E1 -7736.119,E2 -7736.119} C_VEL
LIN {X 0,Y 467.143,Z 385.988,A -85,B 0,C 180,E1 -7736.981,E2 -7736.981} C_VEL
LIN {X 0,Y 466.825,Z 388.792,A -85,B 0,C 180,E1 -7738.273,E2 -7738.273} C_VEL
LIN {X 0,Y 466.79,Z 389.78,A -85,B 0,C 180,E1 -7739.136,E2 -7739.136} C_VEL
LIN {X 0,Y 466.775,Z 390.079,A -85,B 0,C 180,E1 -7739.999,E2 -7739.999} C_VEL
LIN {X 0,Y 466.773,Z 389.698,A -85,B 0,C 180,E1 -7740.862,E2 -7740.862} C_VEL
LIN {X 0,Y 466.793,Z 388.627,A -85,B 0,C 180,E1 -7741.724,E2 -7741.724} C_VEL
LIN {X 0,Y 466.899,Z 386.835,A -85,B 0,C 180,E1 -7742.587,E2 -7742.587} C_VEL
LIN {X 0,Y 467.073,Z 384.284,A -85,B 0,C 180,E1 -7743.449,E2 -7743.449} C_VEL
LIN {X 0,Y 467.318,Z 379.956,A -85,B 0,C 180,E1 -7744.527,E2 -7744.527} C_VEL
LIN {X 0,Y 467.426,Z 373.967,A -85,B 0,C 180,E1 -7745.607,E2 -7745.607} C_VEL
LIN {X 0,Y 467.439,Z 367.783,A -85,B 0,C 180,E1 -7746.473,E2 -7746.473} C_VEL
LIN {X 0,Y 467.64,Z 361.014,A -85,B 0,C 180,E1 -7747.204,E2 -7747.204} C_VEL
LIN {X 0,Y 467.816,Z 353.093,A -85,B 0,C 180,E1 -7747.878,E2 -7747.878} C_VEL
LIN {X 0,Y 467.981,Z 343.61,A -85,B 0,C 180,E1 -7748.473,E2 -7748.473} C_VEL
LIN {X 0,Y 467.708,Z 337.887,A -85,B 0,C 180,E1 -7748.75,E2 -7748.75} C_VEL
LIN {X 0,Y 467.128,Z 333.921,A -85,B 0,C 180,E1 -7748.924,E2 -7748.924} C_VEL
LIN {X 0,Y 467.196,Z 326.327,A -85,B 0,C 180,E1 -7752.156,E2 -7752.156} C_VEL
LIN {X 0,Y 467.195,Z 318.058,A -85,B 0,C 180,E1 -7755.709,E2 -7755.709} C_VEL
LIN {X 0,Y 467.234,Z 311.281,A -85,B 0,C 180,E1 -7758.624,E2 -7758.624} C_VEL
LIN {X 0,Y 467.293,Z 304.333,A -85,B 0,C 180,E1 -7761.62,E2 -7761.62} C_VEL
LIN {X 0,Y 467.353,Z 297.802,A -85,B 0,C 180,E1 -7764.426,E2 -7764.426} C_VEL
LIN {X 0,Y 467.405,Z 290.62,A -85,B 0,C 180,E1 -7767.484,E2 -7767.484} C_VEL
LIN {X 0,Y 467.547,Z 286.249,A -85,B 0,C 180,E1 -7769.364,E2 -7769.364} C_VEL
LIN {X 0,Y 467.567,Z 286.241,A -85,B 0,C 180,E1 -7772.758,E2 -7772.758} C_VEL
LIN {X 0,Y 467.544,Z 286.242,A -85,B 0,C 180,E1 -7775.889,E2 -7775.889} C_VEL
LIN {X 0,Y 467.545,Z 286.247,A -85,B 0,C 180,E1 -7779.146,E2 -7779.146} C_VEL
LIN {X 0,Y 467.559,Z 286.242,A -85,B 0,C 180,E1 -7781.403,E2 -7781.403} C_VEL
LIN {X 0,Y 467.558,Z 286.244,A -85,B 0,C 180,E1 -7785.051,E2 -7785.051} C_VEL
LIN {X 0,Y 467.581,Z 286.239,A -85,B 0,C 180,E1 -7787.439,E2 -7787.439} C_VEL
LIN {X 0,Y 467.574,Z 286.241,A -85,B 0,C 180,E1 -7790.854,E2 -7790.854} C_VEL
LIN {X 0,Y 467.554,Z 286.247,A -85,B 0,C 180,E1 -7794.259,E2 -7794.259} C_VEL
LIN {X 0,Y 467.573,Z 286.242,A -85,B 0,C 180,E1 -7797.32,E2 -7797.32} C_VEL
LIN {X 0,Y 467.568,Z 286.241,A -85,B 0,C 180,E1 -7800.665,E2 -7800.665} C_VEL
LIN {X 0,Y 467.618,Z 286.239,A -85,B 0,C 180,E1 -7803.2,E2 -7803.2} C_VEL
LIN {X 0,Y 467.582,Z 286.24,A -85,B 0,C 180,E1 -7806.467,E2 -7806.467} C_VEL
LIN {X 0,Y 467.613,Z 286.237,A -85,B 0,C 180,E1 -7809.777,E2 -7809.777} C_VEL
LIN {X 0,Y 467.597,Z 286.239,A -85,B 0,C 180,E1 -7812.506,E2 -7812.506} C_VEL
LIN {X 0,Y 467.605,Z 286.236,A -85,B 0,C 180,E1 -7814.574,E2 -7814.574} C_VEL
LIN {X 0,Y 466.913,Z 286.324,A -85,B 0,C 180,E1 -7815.293,E2 -7815.293} C_VEL
LIN {X 0,Y 464.054,Z 286.682,A -85,B 0,C 180,E1 -7816.46,E2 -7816.46} C_VEL
LIN {X 0,Y 461.665,Z 286.977,A -85,B 0,C 180,E1 -7817.402,E2 -7817.402} C_VEL
LIN {X 0,Y 460.66,Z 287.103,A -85,B 0,C 180,E1 -7818.129,E2 -7818.129} C_VEL
LIN {X 0,Y 460.587,Z 287.113,A -85,B 0,C 180,E1 -7818.375,E2 -7818.375} C_VEL
LIN {X 0,Y 460.607,Z 287.108,A -85,B 0,C 180,E1 -7821.223,E2 -7821.223} C_VEL
LIN {X 0,Y 460.669,Z 287.101,A -85,B 0,C 180,E1 -7823.87,E2 -7823.87} C_VEL
LIN {X 0,Y 460.746,Z 287.089,A -85,B 0,C 180,E1 -7827.377,E2 -7827.377} C_VEL
LIN {X 0,Y 460.805,Z 287.089,A -85,B 0,C 180,E1 -7830,E2 -7830} C_VEL
LIN {X 0,Y 460.746,Z 287.089,A -85,B 0,C 180,E1 -7832.623,E2 -7832.623} C_VEL
LIN {X 0,Y 460.669,Z 287.101,A -85,B 0,C 180,E1 -7836.13,E2 -7836.13} C_VEL
LIN {X 0,Y 460.607,Z 287.108,A -85,B 0,C 180,E1 -7838.777,E2 -7838.777} C_VEL
LIN {X 0,Y 460.601,Z 287.109,A -85,B 0,C 180,E1 -7842.445,E2 -7842.445} C_VEL
LIN {X 0,Y 460.588,Z 287.111,A -85,B 0,C 180,E1 -7845.998,E2 -7845.998} C_VEL
LIN {X 0,Y 460.56,Z 287.117,A -85,B 0,C 180,E1 -7848.903,E2 -7848.903} C_VEL
LIN {X 0,Y 460.505,Z 287.122,A -85,B 0,C 180,E1 -7851.486,E2 -7851.486} C_VEL
LIN {X 0,Y 460.532,Z 287.12,A -85,B 0,C 180,E1 -7854.333,E2 -7854.333} C_VEL
LIN {X 0,Y 460.574,Z 287.113,A -85,B 0,C 180,E1 -7857.244,E2 -7857.244} C_VEL
LIN {X 0,Y 460.517,Z 287.122,A -85,B 0,C 180,E1 -7860.24,E2 -7860.24} C_VEL
LIN {X 0,Y 460.52,Z 287.12,A -85,B 0,C 180,E1 -7863.326,E2 -7863.326} C_VEL
LIN {X 0,Y 460.47,Z 287.126,A -85,B 0,C 180,E1 -7866.53,E2 -7866.53} C_VEL
LIN {X 0,Y 460.55,Z 287.117,A -85,B 0,C 180,E1 -7869.861,E2 -7869.861} C_VEL
LIN {X 0,Y 460.505,Z 287.122,A -85,B 0,C 180,E1 -7872.902,E2 -7872.902} C_VEL
LIN {X 0,Y 460.497,Z 287.122,A -85,B 0,C 180,E1 -7875.833,E2 -7875.833} C_VEL
LIN {X 0,Y 460.512,Z 287.124,A -85,B 0,C 180,E1 -7878.989,E2 -7878.989} C_VEL
LIN {X 0,Y 460.491,Z 287.122,A -85,B 0,C 180,E1 -7882.378,E2 -7882.378} C_VEL
LIN {X 0,Y 460.529,Z 287.116,A -85,B 0,C 180,E1 -7885.624,E2 -7885.624} C_VEL
LIN {X 0,Y 460.586,Z 287.114,A -85,B 0,C 180,E1 -7889.26,E2 -7889.26} C_VEL
LIN {X 0,Y 460.627,Z 287.293,A -85,B 0,C 180,E1 -7889.644,E2 -7889.644} C_VEL
LIN {X 0,Y 460.587,Z 292.466,A -85,B 0,C 180,E1 -7892.253,E2 -7892.253} C_VEL
LIN {X 0,Y 460.327,Z 299.38,A -85,B 0,C 180,E1 -7895.657,E2 -7895.657} C_VEL
LIN {X 0,Y 460.231,Z 305.522,A -85,B 0,C 180,E1 -7898.672,E2 -7898.672} C_VEL
LIN {X 0,Y 460.135,Z 310.978,A -85,B 0,C 180,E1 -7901.293,E2 -7901.293} C_VEL
LIN {X 0,Y 459.962,Z 318.662,A -85,B 0,C 180,E1 -7904.946,E2 -7904.946} C_VEL
LIN {X 0,Y 459.872,Z 326.349,A -85,B 0,C 180,E1 -7908.542,E2 -7908.542} C_VEL
LIN {X 0,Y 459.791,Z 330.929,A -85,B 0,C 180,E1 -7910.655,E2 -7910.655} C_VEL
LIN {X 0,Y 461.215,Z 340.69,A -85,B 0,C 180,E1 -7911.126,E2 -7911.126} C_VEL
LIN {X 0,Y 460.995,Z 351.123,A -85,B 0,C 180,E1 -7911.784,E2 -7911.784} C_VEL
LIN {X 0,Y 460.767,Z 360.274,A -85,B 0,C 180,E1 -7912.57,E2 -7912.57} C_VEL
LIN {X 0,Y 460.501,Z 367.986,A -85,B 0,C 180,E1 -7913.429,E2 -7913.429} C_VEL
LIN {X 0,Y 460.435,Z 374.167,A -85,B 0,C 180,E1 -7914.307,E2 -7914.307} C_VEL
LIN {X 0,Y 460.275,Z 380.164,A -85,B 0,C 180,E1 -7915.403,E2 -7915.403} C_VEL
LIN {X 0,Y 460.034,Z 384.626,A -85,B 0,C 180,E1 -7916.498,E2 -7916.498} C_VEL
LIN {X 0,Y 459.85,Z 387.28,A -85,B 0,C 180,E1 -7917.373,E2 -7917.373} C_VEL
LIN {X 0,Y 459.736,Z 389.182,A -85,B 0,C 180,E1 -7918.249,E2 -7918.249} C_VEL
LIN {X 0,Y 459.721,Z 390.377,A -85,B 0,C 180,E1 -7919.125,E2 -7919.125} C_VEL
LIN {X 0,Y 459.729,Z 390.897,A -85,B 0,C 180,E1 -7920.001,E2 -7920.001} C_VEL
LIN {X 0,Y 459.747,Z 390.749,A -85,B 0,C 180,E1 -7920.877,E2 -7920.877} C_VEL
LIN {X 0,Y 459.789,Z 389.933,A -85,B 0,C 180,E1 -7921.753,E2 -7921.753} C_VEL
LIN {X 0,Y 459.887,Z 388.43,A -85,B 0,C 180,E1 -7922.629,E2 -7922.629} C_VEL
LIN {X 0,Y 460.086,Z 386.195,A -85,B 0,C 180,E1 -7923.504,E2 -7923.504} C_VEL
LIN {X 0,Y 460.279,Z 383.174,A -85,B 0,C 180,E1 -7924.38,E2 -7924.38} C_VEL
LIN {X 0,Y 460.583,Z 378.173,A -85,B 0,C 180,E1 -7925.474,E2 -7925.474} C_VEL
LIN {X 0,Y 460.674,Z 373.011,A -85,B 0,C 180,E1 -7926.351,E2 -7926.351} C_VEL
LIN {X 0,Y 460.984,Z 365.309,A -85,B 0,C 180,E1 -7927.37,E2 -7927.37} C_VEL
LIN {X 0,Y 461.388,Z 357.399,A -85,B 0,C 180,E1 -7928.173,E2 -7928.173} C_VEL
LIN {X 0,Y 461.656,Z 348.597,A -85,B 0,C 180,E1 -7928.868,E2 -7928.868} C_VEL
LIN {X 0,Y 461.652,Z 341.561,A -85,B 0,C 180,E1 -7929.31,E2 -7929.31} C_VEL
LIN {X 0,Y 460.046,Z 333.017,A -85,B 0,C 180,E1 -7929.786,E2 -7929.786} C_VEL
LIN {X 0,Y 460.193,Z 327.797,A -85,B 0,C 180,E1 -7932.347,E2 -7932.347} C_VEL
LIN {X 0,Y 460.409,Z 320.578,A -85,B 0,C 180,E1 -7935.949,E2 -7935.949} C_VEL
LIN {X 0,Y 460.611,Z 314.781,A -85,B 0,C 180,E1 -7938.915,E2 -7938.915} C_VEL
LIN {X 0,Y 460.834,Z 308.076,A -85,B 0,C 180,E1 -7942.413,E2 -7942.413} C_VEL
LIN {X 0,Y 461.115,Z 302.836,A -85,B 0,C 180,E1 -7945.263,E2 -7945.263} C_VEL
LIN {X 0,Y 461.408,Z 297.577,A -85,B 0,C 180,E1 -7948.177,E2 -7948.177} C_VEL
LIN {X 0,Y 461.511,Z 294.189,A -85,B 0,C 180,E1 -7950.169,E2 -7950.169} C_VEL
LIN {X 0,Y 461.203,Z 290.908,A -85,B 0,C 180,E1 -7952.233,E2 -7952.233} C_VEL
LIN {X 0,Y 460.529,Z 287.123,A -85,B 0,C 180,E1 -7954.936,E2 -7954.936} C_VEL
LIN {X 0,Y 460.531,Z 287.122,A -85,B 0,C 180,E1 -7958.733,E2 -7958.733} C_VEL
LIN {X 0,Y 460.537,Z 287.122,A -85,B 0,C 180,E1 -7961.603,E2 -7961.603} C_VEL
LIN {X 0,Y 460.519,Z 287.123,A -85,B 0,C 180,E1 -7964.589,E2 -7964.589} C_VEL
LIN {X 0,Y 460.528,Z 287.122,A -85,B 0,C 180,E1 -7967.819,E2 -7967.819} C_VEL
LIN {X 0,Y 460.55,Z 287.12,A -85,B 0,C 180,E1 -7971.103,E2 -7971.103} C_VEL
LIN {X 0,Y 460.508,Z 287.327,A -85,B 0,C 180,E1 -7973.337,E2 -7973.337} C_VEL
LIN {X 0,Y 461.813,Z 292.297,A -85,B 0,C 180,E1 -7975.731,E2 -7975.731} C_VEL
LIN {X 0,Y 463.245,Z 298.573,A -85,B 0,C 180,E1 -7978.168,E2 -7978.168} C_VEL
LIN {X 0,Y 464.733,Z 305.877,A -85,B 0,C 180,E1 -7980.562,E2 -7980.562} C_VEL
LIN {X 0,Y 464.672,Z 309.821,A -85,B 0,C 180,E1 -7981.655,E2 -7981.655} C_VEL
LIN {X 0,Y 463.348,Z 320.8,A -85,B 0,C 180,E1 -7984.387,E2 -7984.387} C_VEL
LIN {X 0,Y 462.257,Z 332.846,A -85,B 0,C 180,E1 -7987.189,E2 -7987.189} C_VEL
LIN {X 0,Y 461.619,Z 343.243,A -85,B 0,C 180,E1 -7989.502,E2 -7989.502} C_VEL
LIN {X 0,Y 460.936,Z 357.304,A -85,B 0,C 180,E1 -7992.474,E2 -7992.474} C_VEL
LIN {X 0,Y 460.56,Z 368.574,A -85,B 0,C 180,E1 -7994.752,E2 -7994.752} C_VEL
LIN {X 0,Y 461.802,Z 380.839,A -85,B 0,C 180,E1 -7995.091,E2 -7995.091} C_VEL
LIN {X 0,Y 462.433,Z 388.964,A -85,B 0,C 180,E1 -7995.393,E2 -7995.393} C_VEL
LIN {X 0,Y 462.108,Z 400.478,A -85,B 0,C 180,E1 -7995.916,E2 -7995.916} C_VEL
LIN {X 0,Y 461.523,Z 413.062,A -85,B 0,C 180,E1 -7996.684,E2 -7996.684} C_VEL
LIN {X 0,Y 461.223,Z 423.727,A -85,B 0,C 180,E1 -7997.52,E2 -7997.52} C_VEL
LIN {X 0,Y 460.666,Z 434.407,A -85,B 0,C 180,E1 -7998.561,E2 -7998.561} C_VEL
LIN {X 0,Y 460.311,Z 443.568,A -85,B 0,C 180,E1 -7999.665,E2 -7999.665} C_VEL
LIN {X 0,Y 460.056,Z 452.497,A -85,B 0,C 180,E1 -8000.991,E2 -8000.991} C_VEL
LIN {X 0,Y 459.877,Z 459.588,A -85,B 0,C 180,E1 -8002.315,E2 -8002.315} C_VEL
LIN {X 0,Y 459.732,Z 466.086,A -85,B 0,C 180,E1 -8003.857,E2 -8003.857} C_VEL
LIN {X 0,Y 459.67,Z 470.322,A -85,B 0,C 180,E1 -8005.176,E2 -8005.176} C_VEL
LIN {X 0,Y 459.772,Z 473.462,A -85,B 0,C 180,E1 -8006.495,E2 -8006.495} C_VEL
LIN {X 0,Y 459.77,Z 474.969,A -85,B 0,C 180,E1 -8007.372,E2 -8007.372} C_VEL
LIN {X 0,Y 459.617,Z 476.685,A -85,B 0,C 180,E1 -8009.124,E2 -8009.124} C_VEL
LIN {X 0,Y 459.622,Z 476.934,A -85,B 0,C 180,E1 -8010,E2 -8010} C_VEL
LIN {X 0,Y 459.614,Z 476.724,A -85,B 0,C 180,E1 -8010.876,E2 -8010.876} C_VEL
LIN {X 0,Y 459.768,Z 475.11,A -85,B 0,C 180,E1 -8012.628,E2 -8012.628} C_VEL
LIN {X 0,Y 459.756,Z 473.628,A -85,B 0,C 180,E1 -8013.506,E2 -8013.506} C_VEL
LIN {X 0,Y 459.659,Z 470.558,A -85,B 0,C 180,E1 -8014.824,E2 -8014.824} C_VEL
LIN {X 0,Y 459.725,Z 466.391,A -85,B 0,C 180,E1 -8016.143,E2 -8016.143} C_VEL
LIN {X 0,Y 459.853,Z 460.995,A -85,B 0,C 180,E1 -8017.464,E2 -8017.464} C_VEL
LIN {X 0,Y 460.013,Z 454.189,A -85,B 0,C 180,E1 -8018.788,E2 -8018.788} C_VEL
LIN {X 0,Y 460.276,Z 445.676,A -85,B 0,C 180,E1 -8020.113,E2 -8020.113} C_VEL
LIN {X 0,Y 460.673,Z 436.868,A -85,B 0,C 180,E1 -8021.216,E2 -8021.216} C_VEL
LIN {X 0,Y 461.055,Z 428.359,A -85,B 0,C 180,E1 -8022.099,E2 -8022.099} C_VEL
LIN {X 0,Y 461.409,Z 417.799,A -85,B 0,C 180,E1 -8022.997,E2 -8022.997} C_VEL
LIN {X 0,Y 461.841,Z 406.598,A -85,B 0,C 180,E1 -8023.755,E2 -8023.755} C_VEL
LIN {X 0,Y 462.259,Z 394.861,A -85,B 0,C 180,E1 -8024.36,E2 -8024.36} C_VEL
LIN {X 0,Y 462.224,Z 385.303,A -85,B 0,C 180,E1 -8024.741,E2 -8024.741} C_VEL
LIN {X 0,Y 460.806,Z 371.511,A -85,B 0,C 180,E1 -8025.14,E2 -8025.14} C_VEL
LIN {X 0,Y 460.564,Z 369.108,A -85,B 0,C 180,E1 -8025.205,E2 -8025.205} C_VEL
LIN {X 0,Y 461.179,Z 353.431,A -85,B 0,C 180,E1 -8028.434,E2 -8028.434} C_VEL
LIN {X 0,Y 462.099,Z 336.115,A -85,B 0,C 180,E1 -8032.061,E2 -8032.061} C_VEL
LIN {X 0,Y 462.978,Z 321.704,A -85,B 0,C 180,E1 -8035.153,E2 -8035.153} C_VEL
LIN {X 0,Y 464.075,Z 307.368,A -85,B 0,C 180,E1 -8038.293,E2 -8038.293} C_VEL
LIN {X 0,Y 464.009,Z 303.215,A -85,B 0,C 180,E1 -8039.24,E2 -8039.24} C_VEL
LIN {X 0,Y 461.743,Z 292.794,A -85,B 0,C 180,E1 -8041.822,E2 -8041.822} C_VEL
LIN {X 0,Y 460.546,Z 287.121,A -85,B 0,C 180,E1 -8043.266,E2 -8043.266} C_VEL
LIN {X 0,Y 460.481,Z 287.128,A -85,B 0,C 180,E1 -8046.529,E2 -8046.529} C_VEL
LIN {X 0,Y 460.537,Z 287.121,A -85,B 0,C 180,E1 -8049.862,E2 -8049.862} C_VEL
LIN {X 0,Y 460.518,Z 287.122,A -85,B 0,C 180,E1 -8052.9,E2 -8052.9} C_VEL
LIN {X 0,Y 460.517,Z 287.124,A -85,B 0,C 180,E1 -8055.83,E2 -8055.83} C_VEL
LIN {X 0,Y 460.536,Z 287.121,A -85,B 0,C 180,E1 -8058.988,E2 -8058.988} C_VEL
LIN {X 0,Y 460.532,Z 287.121,A -85,B 0,C 180,E1 -8061.267,E2 -8061.267} C_VEL
LIN {X 0,Y 460.514,Z 287.125,A -85,B 0,C 180,E1 -8064.554,E2 -8064.554} C_VEL
LIN {X 0,Y 460.534,Z 287.125,A -85,B 0,C 180,E1 -8067.715,E2 -8067.715} C_VEL
LIN {X 0,Y 460.416,Z 287.138,A -85,B 0,C 180,E1 -8071.01,E2 -8071.01} C_VEL
LIN {X 0,Y 460.43,Z 287.211,A -85,B 0,C 180,E1 -8071.26,E2 -8071.26} C_VEL
LIN {X 0,Y 460.468,Z 295.321,A -85,B 0,C 180,E1 -8074.224,E2 -8074.224} C_VEL
LIN {X 0,Y 460.402,Z 302.804,A -85,B 0,C 180,E1 -8077.091,E2 -8077.091} C_VEL
LIN {X 0,Y 460.41,Z 309.745,A -85,B 0,C 180,E1 -8079.912,E2 -8079.912} C_VEL
LIN {X 0,Y 460.324,Z 316.569,A -85,B 0,C 180,E1 -8082.679,E2 -8082.679} C_VEL
LIN {X 0,Y 460.315,Z 323.106,A -85,B 0,C 180,E1 -8085.408,E2 -8085.408} C_VEL
LIN {X 0,Y 460.34,Z 330.505,A -85,B 0,C 180,E1 -8088.551,E2 -8088.551} C_VEL
LIN {X 0,Y 460.298,Z 336.03,A -85,B 0,C 180,E1 -8090.912,E2 -8090.912} C_VEL
LIN {X 0,Y 461.253,Z 342.559,A -85,B 0,C 180,E1 -8091.235,E2 -8091.235} C_VEL
LIN {X 0,Y 461.047,Z 351.843,A -85,B 0,C 180,E1 -8091.783,E2 -8091.783} C_VEL
LIN {X 0,Y 460.886,Z 360.288,A -85,B 0,C 180,E1 -8092.457,E2 -8092.457} C_VEL
LIN {X 0,Y 460.554,Z 367.446,A -85,B 0,C 180,E1 -8093.207,E2 -8093.207} C_VEL
LIN {X 0,Y 460.564,Z 373.998,A -85,B 0,C 180,E1 -8094.087,E2 -8094.087} C_VEL
LIN {X 0,Y 460.355,Z 379.042,A -85,B 0,C 180,E1 -8094.963,E2 -8094.963} C_VEL
LIN {X 0,Y 460.314,Z 383.897,A -85,B 0,C 180,E1 -8096.059,E2 -8096.059} C_VEL
LIN {X 0,Y 460.105,Z 386.723,A -85,B 0,C 180,E1 -8096.934,E2 -8096.934} C_VEL
LIN {X 0,Y 459.861,Z 387.829,A -85,B 0,C 180,E1 -8097.371,E2 -8097.371} C_VEL
LIN {X 0,Y 459.766,Z 389.509,A -85,B 0,C 180,E1 -8098.247,E2 -8098.247} C_VEL
LIN {X 0,Y 459.726,Z 390.477,A -85,B 0,C 180,E1 -8099.123,E2 -8099.123} C_VEL
LIN {X 0,Y 459.708,Z 390.753,A -85,B 0,C 180,E1 -8099.999,E2 -8099.999} C_VEL
LIN {X 0,Y 459.704,Z 390.345,A -85,B 0,C 180,E1 -8100.875,E2 -8100.875} C_VEL
LIN {X 0,Y 459.727,Z 389.245,A -85,B 0,C 180,E1 -8101.751,E2 -8101.751} C_VEL
LIN {X 0,Y 460.056,Z 386.24,A -85,B 0,C 180,E1 -8103.064,E2 -8103.064} C_VEL
LIN {X 0,Y 460.12,Z 383.291,A -85,B 0,C 180,E1 -8103.94,E2 -8103.94} C_VEL
LIN {X 0,Y 460.286,Z 378.238,A -85,B 0,C 180,E1 -8105.036,E2 -8105.036} C_VEL
LIN {X 0,Y 460.433,Z 373.023,A -85,B 0,C 180,E1 -8105.913,E2 -8105.913} C_VEL
LIN {X 0,Y 460.47,Z 366.258,A -85,B 0,C 180,E1 -8106.792,E2 -8106.792} C_VEL
LIN {X 0,Y 460.703,Z 359.069,A -85,B 0,C 180,E1 -8107.526,E2 -8107.526} C_VEL
LIN {X 0,Y 460.847,Z 350.124,A -85,B 0,C 180,E1 -8108.219,E2 -8108.219} C_VEL
LIN {X 0,Y 460.944,Z 341.556,A -85,B 0,C 180,E1 -8108.714,E2 -8108.714} C_VEL
LIN {X 0,Y 460.077,Z 334.416,A -85,B 0,C 180,E1 -8109.062,E2 -8109.062} C_VEL
LIN {X 0,Y 460.138,Z 326.706,A -85,B 0,C 180,E1 -8112.346,E2 -8112.346} C_VEL
LIN {X 0,Y 460.134,Z 318.331,A -85,B 0,C 180,E1 -8115.956,E2 -8115.956} C_VEL
LIN {X 0,Y 460.211,Z 310.985,A -85,B 0,C 180,E1 -8119.12,E2 -8119.12} C_VEL
LIN {X 0,Y 460.25,Z 304.389,A -85,B 0,C 180,E1 -8121.968,E2 -8121.968} C_VEL
LIN {X 0,Y 460.317,Z 296.613,A -85,B 0,C 180,E1 -8125.307,E2 -8125.307} C_VEL
LIN {X 0,Y 460.431,Z 288.56,A -85,B 0,C 180,E1 -8128.737,E2 -8128.737} C_VEL
LIN {X 0,Y 460.49,Z 287.128,A -85,B 0,C 180,E1 -8129.354,E2 -8129.354} C_VEL
LIN {X 0,Y 460.508,Z 287.118,A -85,B 0,C 180,E1 -8132.284,E2 -8132.284} C_VEL
LIN {X 0,Y 460.5,Z 287.123,A -85,B 0,C 180,E1 -8135.445,E2 -8135.445} C_VEL
LIN {X 0,Y 460.522,Z 287.123,A -85,B 0,C 180,E1 -8138.894,E2 -8138.894} C_VEL
LIN {X 0,Y 460.495,Z 287.122,A -85,B 0,C 180,E1 -8142.182,E2 -8142.182} C_VEL
LIN {X 0,Y 460.506,Z 287.121,A -85,B 0,C 180,E1 -8145.41,E2 -8145.41} C_VEL
LIN {X 0,Y 460.524,Z 287.122,A -85,B 0,C 180,E1 -8148.396,E2 -8148.396} C_VEL
LIN {X 0,Y 460.518,Z 287.119,A -85,B 0,C 180,E1 -8151.266,E2 -8151.266} C_VEL
LIN {X 0,Y 460.505,Z 287.123,A -85,B 0,C 180,E1 -8154.554,E2 -8154.554} C_VEL
LIN {X 0,Y 460.523,Z 287.121,A -85,B 0,C 180,E1 -8157.715,E2 -8157.715} C_VEL
LIN {X 0,Y 460.537,Z 287.117,A -85,B 0,C 180,E1 -8160.769,E2 -8160.769} C_VEL
LIN {X 0,Y 460.558,Z 287.117,A -85,B 0,C 180,E1 -8163.734,E2 -8163.734} C_VEL
LIN {X 0,Y 460.535,Z 287.118,A -85,B 0,C 180,E1 -8166.623,E2 -8166.623} C_VEL
LIN {X 0,Y 460.541,Z 287.118,A -85,B 0,C 180,E1 -8169.452,E2 -8169.452} C_VEL
LIN {X 0,Y 460.547,Z 287.116,A -85,B 0,C 180,E1 -8172.23,E2 -8172.23} C_VEL
LIN {X 0,Y 460.553,Z 287.117,A -85,B 0,C 180,E1 -8174.964,E2 -8174.964} C_VEL
LIN {X 0,Y 460.587,Z 287.113,A -85,B 0,C 180,E1 -8178.375,E2 -8178.375} C_VEL
LIN {X 0,Y 459.937,Z 287.199,A -85,B 0,C 180,E1 -8179.105,E2 -8179.105} C_VEL
LIN {X 0,Y 457.063,Z 287.556,A -85,B 0,C 180,E1 -8180.29,E2 -8180.29} C_VEL
LIN {X 0,Y 454.645,Z 287.853,A -85,B 0,C 180,E1 -8181.246,E2 -8181.246} C_VEL
LIN {X 0,Y 453.645,Z 287.977,A -85,B 0,C 180,E1 -8181.985,E2 -8181.985} C_VEL
LIN {X 0,Y 453.584,Z 287.984,A -85,B 0,C 180,E1 -8182.235,E2 -8182.235} C_VEL
LIN {X 0,Y 453.646,Z 287.976,A -85,B 0,C 180,E1 -8184.666,E2 -8184.666} C_VEL
LIN {X 0,Y 453.674,Z 287.975,A -85,B 0,C 180,E1 -8188.225,E2 -8188.225} C_VEL
LIN {X 0,Y 453.775,Z 287.964,A -85,B 0,C 180,E1 -8190,E2 -8190} C_VEL
LIN {X 0,Y 453.693,Z 287.968,A -85,B 0,C 180,E1 -8192.664,E2 -8192.664} C_VEL
LIN {X 0,Y 453.635,Z 287.977,A -85,B 0,C 180,E1 -8196.226,E2 -8196.226} C_VEL
LIN {X 0,Y 453.573,Z 287.985,A -85,B 0,C 180,E1 -8198.914,E2 -8198.914} C_VEL
LIN {X 0,Y 453.551,Z 287.987,A -85,B 0,C 180,E1 -8202.529,E2 -8202.529} C_VEL
LIN {X 0,Y 453.533,Z 287.99,A -85,B 0,C 180,E1 -8206.196,E2 -8206.196} C_VEL
LIN {X 0,Y 453.509,Z 287.996,A -85,B 0,C 180,E1 -8209.042,E2 -8209.042} C_VEL
LIN {X 0,Y 453.465,Z 287.998,A -85,B 0,C 180,E1 -8211.837,E2 -8211.837} C_VEL
LIN {X 0,Y 453.504,Z 287.996,A -85,B 0,C 180,E1 -8214.735,E2 -8214.735} C_VEL
LIN {X 0,Y 453.529,Z 287.993,A -85,B 0,C 180,E1 -8217.962,E2 -8217.962} C_VEL
LIN {X 0,Y 453.473,Z 287.999,A -85,B 0,C 180,E1 -8220.76,E2 -8220.76} C_VEL
LIN {X 0,Y 453.469,Z 288,A -85,B 0,C 180,E1 -8223.914,E2 -8223.914} C_VEL
LIN {X 0,Y 453.462,Z 287.999,A -85,B 0,C 180,E1 -8227.189,E2 -8227.189} C_VEL
LIN {X 0,Y 453.508,Z 287.997,A -85,B 0,C 180,E1 -8229.448,E2 -8229.448} C_VEL
LIN {X 0,Y 453.455,Z 288.001,A -85,B 0,C 180,E1 -8232.996,E2 -8232.996} C_VEL
LIN {X 0,Y 453.452,Z 288,A -85,B 0,C 180,E1 -8235.779,E2 -8235.779} C_VEL
LIN {X 0,Y 453.463,Z 288,A -85,B 0,C 180,E1 -8239.39,E2 -8239.39} C_VEL
LIN {X 0,Y 453.442,Z 288.005,A -85,B 0,C 180,E1 -8242.811,E2 -8242.811} C_VEL
LIN {X 0,Y 453.46,Z 287.997,A -85,B 0,C 180,E1 -8246.088,E2 -8246.088} C_VEL
LIN {X 0,Y 453.545,Z 288.008,A -85,B 0,C 180,E1 -8249.503,E2 -8249.503} C_VEL
LIN {X 0,Y 453.559,Z 292.974,A -85,B 0,C 180,E1 -8252.035,E2 -8252.035} C_VEL
LIN {X 0,Y 453.305,Z 299.42,A -85,B 0,C 180,E1 -8255.255,E2 -8255.255} C_VEL
LIN {X 0,Y 453.177,Z 306.029,A -85,B 0,C 180,E1 -8258.513,E2 -8258.513} C_VEL
LIN {X 0,Y 453.015,Z 313.052,A -85,B 0,C 180,E1 -8261.926,E2 -8261.926} C_VEL
LIN {X 0,Y 452.891,Z 318.854,A -85,B 0,C 180,E1 -8264.705,E2 -8264.705} C_VEL
LIN {X 0,Y 452.818,Z 326.596,A -85,B 0,C 180,E1 -8268.361,E2 -8268.361} C_VEL
LIN {X 0,Y 452.755,Z 331.256,A -85,B 0,C 180,E1 -8270.508,E2 -8270.508} C_VEL
LIN {X 0,Y 454.251,Z 342.088,A -85,B 0,C 180,E1 -8271.045,E2 -8271.045} C_VEL
LIN {X 0,Y 453.979,Z 351.491,A -85,B 0,C 180,E1 -8271.656,E2 -8271.656} C_VEL
LIN {X 0,Y 453.783,Z 360.098,A -85,B 0,C 180,E1 -8272.397,E2 -8272.397} C_VEL
LIN {X 0,Y 453.459,Z 368.424,A -85,B 0,C 180,E1 -8273.326,E2 -8273.326} C_VEL
LIN {X 0,Y 453.407,Z 374.639,A -85,B 0,C 180,E1 -8274.219,E2 -8274.219} C_VEL
LIN {X 0,Y 453.233,Z 380.682,A -85,B 0,C 180,E1 -8275.332,E2 -8275.332} C_VEL
LIN {X 0,Y 452.996,Z 385.19,A -85,B 0,C 180,E1 -8276.443,E2 -8276.443} C_VEL
LIN {X 0,Y 452.8,Z 387.875,A -85,B 0,C 180,E1 -8277.332,E2 -8277.332} C_VEL
LIN {X 0,Y 452.672,Z 389.808,A -85,B 0,C 180,E1 -8278.222,E2 -8278.222} C_VEL
LIN {X 0,Y 452.653,Z 391.032,A -85,B 0,C 180,E1 -8279.112,E2 -8279.112} C_VEL
LIN {X 0,Y 452.662,Z 391.578,A -85,B 0,C 180,E1 -8280.001,E2 -8280.001} C_VEL
LIN {X 0,Y 452.684,Z 391.457,A -85,B 0,C 180,E1 -8280.891,E2 -8280.891} C_VEL
LIN {X 0,Y 452.732,Z 390.671,A -85,B 0,C 180,E1 -8281.78,E2 -8281.78} C_VEL
LIN {X 0,Y 452.837,Z 389.203,A -85,B 0,C 180,E1 -8282.67,E2 -8282.67} C_VEL
LIN {X 0,Y 453.05,Z 387.01,A -85,B 0,C 180,E1 -8283.559,E2 -8283.559} C_VEL
LIN {X 0,Y 453.256,Z 384.045,A -85,B 0,C 180,E1 -8284.448,E2 -8284.448} C_VEL
LIN {X 0,Y 453.576,Z 379.118,A -85,B 0,C 180,E1 -8285.558,E2 -8285.558} C_VEL
LIN {X 0,Y 453.794,Z 372.564,A -85,B 0,C 180,E1 -8286.671,E2 -8286.671} C_VEL
LIN {X 0,Y 454.08,Z 365.782,A -85,B 0,C 180,E1 -8287.56,E2 -8287.56} C_VEL
LIN {X 0,Y 454.518,Z 357.054,A -85,B 0,C 180,E1 -8288.448,E2 -8288.448} C_VEL
LIN {X 0,Y 454.803,Z 348.555,A -85,B 0,C 180,E1 -8289.115,E2 -8289.115} C_VEL
LIN {X 0,Y 454.848,Z 343.298,A -85,B 0,C 180,E1 -8289.45,E2 -8289.45} C_VEL
LIN {X 0,Y 453.052,Z 333.497,A -85,B 0,C 180,E1 -8290.023,E2 -8290.023} C_VEL
LIN {X 0,Y 453.168,Z 328.428,A -85,B 0,C 180,E1 -8292.541,E2 -8292.541} C_VEL
LIN {X 0,Y 453.406,Z 321.226,A -85,B 0,C 180,E1 -8296.202,E2 -8296.202} C_VEL
LIN {X 0,Y 453.611,Z 315.669,A -85,B 0,C 180,E1 -8299.073,E2 -8299.073} C_VEL
LIN {X 0,Y 453.809,Z 310.473,A -85,B 0,C 180,E1 -8301.82,E2 -8301.82} C_VEL
LIN {X 0,Y 454.091,Z 305.299,A -85,B 0,C 180,E1 -8304.702,E2 -8304.702} C_VEL
LIN {X 0,Y 454.421,Z 300.074,A -85,B 0,C 180,E1 -8307.645,E2 -8307.645} C_VEL
LIN {X 0,Y 454.625,Z 296.075,A -85,B 0,C 180,E1 -8310.037,E2 -8310.037} C_VEL
LIN {X 0,Y 454.237,Z 291.903,A -85,B 0,C 180,E1 -8312.788,E2 -8312.788} C_VEL
LIN {X 0,Y 453.461,Z 288.003,A -85,B 0,C 180,E1 -8315.809,E2 -8315.809} C_VEL
LIN {X 0,Y 453.5,Z 287.998,A -85,B 0,C 180,E1 -8319.207,E2 -8319.207} C_VEL
LIN {X 0,Y 453.482,Z 288,A -85,B 0,C 180,E1 -8321.935,E2 -8321.935} C_VEL
LIN {X 0,Y 453.489,Z 287.999,A -85,B 0,C 180,E1 -8325.472,E2 -8325.472} C_VEL
LIN {X 0,Y 453.484,Z 288,A -85,B 0,C 180,E1 -8328.21,E2 -8328.21} C_VEL
LIN {X 0,Y 453.499,Z 287.998,A -85,B 0,C 180,E1 -8330.794,E2 -8330.794} C_VEL
LIN {X 0,Y 453.469,Z 288.052,A -85,B 0,C 180,E1 -8332.225,E2 -8332.225} C_VEL
LIN {X 0,Y 454.516,Z 292.23,A -85,B 0,C 180,E1 -8334.561,E2 -8334.561} C_VEL
LIN {X 0,Y 455.83,Z 297.544,A -85,B 0,C 180,E1 -8336.891,E2 -8336.891} C_VEL
LIN {X 0,Y 457.386,Z 304.837,A -85,B 0,C 180,E1 -8339.531,E2 -8339.531} C_VEL
LIN {X 0,Y 458.03,Z 309.538,A -85,B 0,C 180,E1 -8341,E2 -8341} C_VEL
LIN {X 0,Y 456.837,Z 319.121,A -85,B 0,C 180,E1 -8343.504,E2 -8343.504} C_VEL
LIN {X 0,Y 455.587,Z 330.884,A -85,B 0,C 180,E1 -8346.354,E2 -8346.354} C_VEL
LIN {X 0,Y 454.802,Z 342.096,A -85,B 0,C 180,E1 -8348.944,E2 -8348.944} C_VEL
LIN {X 0,Y 453.934,Z 357.055,A -85,B 0,C 180,E1 -8352.195,E2 -8352.195} C_VEL
LIN {X 0,Y 453.528,Z 368.09,A -85,B 0,C 180,E1 -8354.509,E2 -8354.509} C_VEL
LIN {X 0,Y 454.859,Z 381.013,A -85,B 0,C 180,E1 -8354.886,E2 -8354.886} C_VEL
LIN {X 0,Y 455.464,Z 390.311,A -85,B 0,C 180,E1 -8355.25,E2 -8355.25} C_VEL
LIN {X 0,Y 454.989,Z 403.702,A -85,B 0,C 180,E1 -8355.92,E2 -8355.92} C_VEL
LIN {X 0,Y 454.468,Z 415.064,A -85,B 0,C 180,E1 -8356.673,E2 -8356.673} C_VEL
LIN {X 0,Y 454.124,Z 426.012,A -85,B 0,C 180,E1 -8357.6,E2 -8357.6} C_VEL
LIN {X 0,Y 453.593,Z 435.697,A -85,B 0,C 180,E1 -8358.606,E2 -8358.606} C_VEL
LIN {X 0,Y 453.219,Z 444.531,A -85,B 0,C 180,E1 -8359.728,E2 -8359.728} C_VEL
LIN {X 0,Y 452.959,Z 453.075,A -85,B 0,C 180,E1 -8361.074,E2 -8361.074} C_VEL
LIN {X 0,Y 452.784,Z 459.948,A -85,B 0,C 180,E1 -8362.419,E2 -8362.419} C_VEL
LIN {X 0,Y 452.659,Z 465.416,A -85,B 0,C 180,E1 -8363.761,E2 -8363.761} C_VEL
LIN {X 0,Y 452.6,Z 469.657,A -85,B 0,C 180,E1 -8365.101,E2 -8365.101} C_VEL
LIN {X 0,Y 452.699,Z 472.8,A -85,B 0,C 180,E1 -8366.44,E2 -8366.44} C_VEL
LIN {X 0,Y 452.716,Z 474.309,A -85,B 0,C 180,E1 -8367.331,E2 -8367.331} C_VEL
LIN {X 0,Y 452.549,Z 476.026,A -85,B 0,C 180,E1 -8369.11,E2 -8369.11} C_VEL
LIN {X 0,Y 452.554,Z 476.271,A -85,B 0,C 180,E1 -8370,E2 -8370} C_VEL
LIN {X 0,Y 452.546,Z 476.058,A -85,B 0,C 180,E1 -8370.89,E2 -8370.89} C_VEL
LIN {X 0,Y 452.596,Z 475.447,A -85,B 0,C 180,E1 -8371.78,E2 -8371.78} C_VEL
LIN {X 0,Y 452.712,Z 474.436,A -85,B 0,C 180,E1 -8372.669,E2 -8372.669} C_VEL
LIN {X 0,Y 452.683,Z 472.937,A -85,B 0,C 180,E1 -8373.56,E2 -8373.56} C_VEL
LIN {X 0,Y 452.591,Z 469.847,A -85,B 0,C 180,E1 -8374.899,E2 -8374.899} C_VEL
LIN {X 0,Y 452.693,Z 464.757,A -85,B 0,C 180,E1 -8376.486,E2 -8376.486} C_VEL
LIN {X 0,Y 452.836,Z 458.122,A -85,B 0,C 180,E1 -8378.029,E2 -8378.029} C_VEL
LIN {X 0,Y 453.017,Z 450.711,A -85,B 0,C 180,E1 -8379.375,E2 -8379.375} C_VEL
LIN {X 0,Y 453.295,Z 443.131,A -85,B 0,C 180,E1 -8380.497,E2 -8380.497} C_VEL
LIN {X 0,Y 453.672,Z 433.914,A -85,B 0,C 180,E1 -8381.618,E2 -8381.618} C_VEL
LIN {X 0,Y 454.189,Z 423.737,A -85,B 0,C 180,E1 -8382.615,E2 -8382.615} C_VEL
LIN {X 0,Y 454.596,Z 412.143,A -85,B 0,C 180,E1 -8383.523,E2 -8383.523} C_VEL
LIN {X 0,Y 455.096,Z 400.141,A -85,B 0,C 180,E1 -8384.248,E2 -8384.248} C_VEL
LIN {X 0,Y 455.362,Z 387.141,A -85,B 0,C 180,E1 -8384.825,E2 -8384.825} C_VEL
LIN {X 0,Y 454.066,Z 373.81,A -85,B 0,C 180,E1 -8385.256,E2 -8385.256} C_VEL
LIN {X 0,Y 453.516,Z 368.844,A -85,B 0,C 180,E1 -8385.385,E2 -8385.385} C_VEL
LIN {X 0,Y 454.139,Z 354.042,A -85,B 0,C 180,E1 -8388.497,E2 -8388.497} C_VEL
LIN {X 0,Y 455.068,Z 337.284,A -85,B 0,C 180,E1 -8392.083,E2 -8392.083} C_VEL
LIN {X 0,Y 456.035,Z 322.45,A -85,B 0,C 180,E1 -8395.319,E2 -8395.319} C_VEL
LIN {X 0,Y 457.17,Z 308.393,A -85,B 0,C 180,E1 -8398.461,E2 -8398.461} C_VEL
LIN {X 0,Y 457.256,Z 305.69,A -85,B 0,C 180,E1 -8399.082,E2 -8399.082} C_VEL
LIN {X 0,Y 454.916,Z 294.76,A -85,B 0,C 180,E1 -8401.82,E2 -8401.82} C_VEL
LIN {X 0,Y 453.485,Z 288,A -85,B 0,C 180,E1 -8403.618,E2 -8403.618} C_VEL
LIN {X 0,Y 453.458,Z 288.003,A -85,B 0,C 180,E1 -8406.299,E2 -8406.299} C_VEL
LIN {X 0,Y 453.495,Z 287.997,A -85,B 0,C 180,E1 -8409.449,E2 -8409.449} C_VEL
LIN {X 0,Y 453.482,Z 288,A -85,B 0,C 180,E1 -8411.934,E2 -8411.934} C_VEL
LIN {X 0,Y 453.492,Z 287.997,A -85,B 0,C 180,E1 -8415.47,E2 -8415.47} C_VEL
LIN {X 0,Y 453.484,Z 287.998,A -85,B 0,C 180,E1 -8418.209,E2 -8418.209} C_VEL
LIN {X 0,Y 453.515,Z 287.995,A -85,B 0,C 180,E1 -8420.79,E2 -8420.79} C_VEL
LIN {X 0,Y 453.459,Z 288.002,A -85,B 0,C 180,E1 -8423.917,E2 -8423.917} C_VEL
LIN {X 0,Y 453.484,Z 288.003,A -85,B 0,C 180,E1 -8427.15,E2 -8427.15} C_VEL
LIN {X 0,Y 453.415,Z 288.009,A -85,B 0,C 180,E1 -8430.263,E2 -8430.263} C_VEL
LIN {X 0,Y 453.409,Z 288.172,A -85,B 0,C 180,E1 -8431.09,E2 -8431.09} C_VEL
LIN {X 0,Y 453.482,Z 294.15,A -85,B 0,C 180,E1 -8433.291,E2 -8433.291} C_VEL
LIN {X 0,Y 453.457,Z 301.879,A -85,B 0,C 180,E1 -8436.235,E2 -8436.235} C_VEL
LIN {X 0,Y 453.427,Z 310.232,A -85,B 0,C 180,E1 -8439.588,E2 -8439.588} C_VEL
LIN {X 0,Y 453.342,Z 318.186,A -85,B 0,C 180,E1 -8442.868,E2 -8442.868} C_VEL
LIN {X 0,Y 453.303,Z 325.879,A -85,B 0,C 180,E1 -8446.094,E2 -8446.094} C_VEL
LIN {X 0,Y 453.327,Z 332.267,A -85,B 0,C 180,E1 -8448.825,E2 -8448.825} C_VEL
LIN {X 0,Y 453.265,Z 336.852,A -85,B 0,C 180,E1 -8450.756,E2 -8450.756} C_VEL
LIN {X 0,Y 454.3,Z 343.892,A -85,B 0,C 180,E1 -8451.1,E2 -8451.1} C_VEL
LIN {X 0,Y 454.088,Z 353.017,A -85,B 0,C 180,E1 -8451.656,E2 -8451.656} C_VEL
LIN {X 0,Y 453.928,Z 361.238,A -85,B 0,C 180,E1 -8452.333,E2 -8452.333} C_VEL
LIN {X 0,Y 453.582,Z 368.422,A -85,B 0,C 180,E1 -8453.102,E2 -8453.102} C_VEL
LIN {X 0,Y 453.558,Z 374.886,A -85,B 0,C 180,E1 -8453.995,E2 -8453.995} C_VEL
LIN {X 0,Y 453.335,Z 379.882,A -85,B 0,C 180,E1 -8454.885,E2 -8454.885} C_VEL
LIN {X 0,Y 453.288,Z 384.686,A -85,B 0,C 180,E1 -8455.998,E2 -8455.998} C_VEL
LIN {X 0,Y 453.069,Z 387.476,A -85,B 0,C 180,E1 -8456.887,E2 -8456.887} C_VEL
LIN {X 0,Y 452.811,Z 388.578,A -85,B 0,C 180,E1 -8457.33,E2 -8457.33} C_VEL
LIN {X 0,Y 452.707,Z 390.234,A -85,B 0,C 180,E1 -8458.22,E2 -8458.22} C_VEL
LIN {X 0,Y 452.662,Z 391.174,A -85,B 0,C 180,E1 -8459.109,E2 -8459.109} C_VEL
LIN {X 0,Y 452.641,Z 391.425,A -85,B 0,C 180,E1 -8459.999,E2 -8459.999} C_VEL
LIN {X 0,Y 452.635,Z 390.991,A -85,B 0,C 180,E1 -8460.888,E2 -8460.888} C_VEL
LIN {X 0,Y 452.664,Z 389.861,A -85,B 0,C 180,E1 -8461.778,E2 -8461.778} C_VEL
LIN {X 0,Y 452.986,Z 386.821,A -85,B 0,C 180,E1 -8463.112,E2 -8463.112} C_VEL
LIN {X 0,Y 453.084,Z 383.826,A -85,B 0,C 180,E1 -8464.001,E2 -8464.001} C_VEL
LIN {X 0,Y 453.243,Z 378.717,A -85,B 0,C 180,E1 -8465.114,E2 -8465.114} C_VEL
LIN {X 0,Y 453.402,Z 373.456,A -85,B 0,C 180,E1 -8466.005,E2 -8466.005} C_VEL
LIN {X 0,Y 453.456,Z 366.22,A -85,B 0,C 180,E1 -8466.942,E2 -8466.942} C_VEL
LIN {X 0,Y 453.693,Z 359.004,A -85,B 0,C 180,E1 -8467.676,E2 -8467.676} C_VEL
LIN {X 0,Y 453.826,Z 350.266,A -85,B 0,C 180,E1 -8468.347,E2 -8468.347} C_VEL
LIN {X 0,Y 453.915,Z 341.56,A -85,B 0,C 180,E1 -8468.85,E2 -8468.85} C_VEL
LIN {X 0,Y 452.984,Z 335.039,A -85,B 0,C 180,E1 -8469.149,E2 -8469.149} C_VEL
LIN {X 0,Y 453.083,Z 327.082,A -85,B 0,C 180,E1 -8472.541,E2 -8472.541} C_VEL
LIN {X 0,Y 453.097,Z 318.553,A -85,B 0,C 180,E1 -8476.211,E2 -8476.211} C_VEL
LIN {X 0,Y 453.176,Z 310.999,A -85,B 0,C 180,E1 -8479.476,E2 -8479.476} C_VEL
LIN {X 0,Y 453.199,Z 304.393,A -85,B 0,C 180,E1 -8482.328,E2 -8482.328} C_VEL
LIN {X 0,Y 453.269,Z 297.688,A -85,B 0,C 180,E1 -8485.237,E2 -8485.237} C_VEL
LIN {X 0,Y 453.345,Z 291.387,A -85,B 0,C 180,E1 -8487.914,E2 -8487.914} C_VEL
LIN {X 0,Y 453.466,Z 288.003,A -85,B 0,C 180,E1 -8489.412,E2 -8489.412} C_VEL
LIN {X 0,Y 453.467,Z 287.998,A -85,B 0,C 180,E1 -8492.848,E2 -8492.848} C_VEL
LIN {X 0,Y 453.445,Z 287.999,A -85,B 0,C 180,E1 -8496.082,E2 -8496.082} C_VEL
LIN {X 0,Y 453.453,Z 288,A -85,B 0,C 180,E1 -8499.452,E2 -8499.452} C_VEL
LIN {X 0,Y 453.449,Z 287.999,A -85,B 0,C 180,E1 -8501.931,E2 -8501.931} C_VEL
LIN {X 0,Y 453.476,Z 287.996,A -85,B 0,C 180,E1 -8505.47,E2 -8505.47} C_VEL
LIN {X 0,Y 453.471,Z 287.999,A -85,B 0,C 180,E1 -8508.208,E2 -8508.208} C_VEL
LIN {X 0,Y 453.507,Z 287.994,A -85,B 0,C 180,E1 -8510.789,E2 -8510.789} C_VEL
LIN {X 0,Y 453.448,Z 288.002,A -85,B 0,C 180,E1 -8513.916,E2 -8513.916} C_VEL
LIN {X 0,Y 453.474,Z 287.998,A -85,B 0,C 180,E1 -8517.15,E2 -8517.15} C_VEL
LIN {X 0,Y 453.504,Z 287.995,A -85,B 0,C 180,E1 -8520.27,E2 -8520.27} C_VEL
LIN {X 0,Y 453.504,Z 287.996,A -85,B 0,C 180,E1 -8523.294,E2 -8523.294} C_VEL
LIN {X 0,Y 453.493,Z 287.995,A -85,B 0,C 180,E1 -8526.238,E2 -8526.238} C_VEL
LIN {X 0,Y 453.472,Z 288,A -85,B 0,C 180,E1 -8529.117,E2 -8529.117} C_VEL
LIN {X 0,Y 453.5,Z 287.994,A -85,B 0,C 180,E1 -8531.944,E2 -8531.944} C_VEL
LIN {X 0,Y 453.528,Z 287.994,A -85,B 0,C 180,E1 -8534.726,E2 -8534.726} C_VEL
LIN {X 0,Y 453.546,Z 287.991,A -85,B 0,C 180,E1 -8538.379,E2 -8538.379} C_VEL
LIN {X 0,Y 453.572,Z 287.984,A -85,B 0,C 180,E1 -8541.086,E2 -8541.086} C_VEL
LIN {X 0,Y 453.584,Z 287.984,A -85,B 0,C 180,E1 -8542.235,E2 -8542.235} C_VEL
LIN {X 0,Y 452.956,Z 288.065,A -85,B 0,C 180,E1 -8542.977,E2 -8542.977} C_VEL
LIN {X 0,Y 450.048,Z 288.428,A -85,B 0,C 180,E1 -8544.181,E2 -8544.181} C_VEL
LIN {X 0,Y 447.56,Z 288.733,A -85,B 0,C 180,E1 -8545.152,E2 -8545.152} C_VEL
LIN {X 0,Y 446.497,Z 288.868,A -85,B 0,C 180,E1 -8545.903,E2 -8545.903} C_VEL
LIN {X 0,Y 446.415,Z 288.876,A -85,B 0,C 180,E1 -8546.158,E2 -8546.158} C_VEL
LIN {X 0,Y 446.644,Z 288.851,A -85,B 0,C 180,E1 -8548.197,E2 -8548.197} C_VEL
LIN {X 0,Y 446.724,Z 288.843,A -85,B 0,C 180,E1 -8550,E2 -8550} C_VEL
LIN {X 0,Y 446.643,Z 288.846,A -85,B 0,C 180,E1 -8552.706,E2 -8552.706} C_VEL
LIN {X 0,Y 446.603,Z 288.852,A -85,B 0,C 180,E1 -8556.324,E2 -8556.324} C_VEL
LIN {X 0,Y 446.52,Z 288.863,A -85,B 0,C 180,E1 -8559.056,E2 -8559.056} C_VEL
LIN {X 0,Y 446.509,Z 288.865,A -85,B 0,C 180,E1 -8562.73,E2 -8562.73} C_VEL
LIN {X 0,Y 446.484,Z 288.868,A -85,B 0,C 180,E1 -8566.228,E2 -8566.228} C_VEL
LIN {X 0,Y 446.458,Z 288.874,A -85,B 0,C 180,E1 -8569.304,E2 -8569.304} C_VEL
LIN {X 0,Y 446.407,Z 288.879,A -85,B 0,C 180,E1 -8572.2,E2 -8572.2} C_VEL
LIN {X 0,Y 446.448,Z 288.874,A -85,B 0,C 180,E1 -8575.153,E2 -8575.153} C_VEL
LIN {X 0,Y 446.474,Z 288.871,A -85,B 0,C 180,E1 -8578.18,E2 -8578.18} C_VEL
LIN {X 0,Y 446.41,Z 288.878,A -85,B 0,C 180,E1 -8581.301,E2 -8581.301} C_VEL
LIN {X 0,Y 446.422,Z 288.878,A -85,B 0,C 180,E1 -8584.524,E2 -8584.524} C_VEL
LIN {X 0,Y 446.422,Z 288.877,A -85,B 0,C 180,E1 -8588.083,E2 -8588.083} C_VEL
LIN {X 0,Y 446.419,Z 288.876,A -85,B 0,C 180,E1 -8590.919,E2 -8590.919} C_VEL
LIN {X 0,Y 446.392,Z 288.88,A -85,B 0,C 180,E1 -8593.847,E2 -8593.847} C_VEL
LIN {X 0,Y 446.39,Z 288.879,A -85,B 0,C 180,E1 -8596.405,E2 -8596.405} C_VEL
LIN {X 0,Y 446.398,Z 288.883,A -85,B 0,C 180,E1 -8599.087,E2 -8599.087} C_VEL
LIN {X 0,Y 446.398,Z 288.877,A -85,B 0,C 180,E1 -8602.122,E2 -8602.122} C_VEL
LIN {X 0,Y 446.415,Z 288.874,A -85,B 0,C 180,E1 -8605.478,E2 -8605.478} C_VEL
LIN {X 0,Y 446.538,Z 288.864,A -85,B 0,C 180,E1 -8609.237,E2 -8609.237} C_VEL
LIN {X 0,Y 446.536,Z 288.974,A -85,B 0,C 180,E1 -8609.499,E2 -8609.499} C_VEL
LIN {X 0,Y 446.517,Z 293.509,A -85,B 0,C 180,E1 -8611.825,E2 -8611.825} C_VEL
LIN {X 0,Y 446.292,Z 299.461,A -85,B 0,C 180,E1 -8614.839,E2 -8614.839} C_VEL
LIN {X 0,Y 446.135,Z 306.488,A -85,B 0,C 180,E1 -8618.347,E2 -8618.347} C_VEL
LIN {X 0,Y 445.973,Z 313.189,A -85,B 0,C 180,E1 -8621.63,E2 -8621.63} C_VEL
LIN {X 0,Y 445.828,Z 319.043,A -85,B 0,C 180,E1 -8624.457,E2 -8624.457} C_VEL
LIN {X 0,Y 445.77,Z 326.833,A -85,B 0,C 180,E1 -8628.174,E2 -8628.174} C_VEL
LIN {X 0,Y 445.681,Z 331.664,A -85,B 0,C 180,E1 -8630.356,E2 -8630.356} C_VEL
LIN {X 0,Y 447.236,Z 342.45,A -85,B 0,C 180,E1 -8630.903,E2 -8630.903} C_VEL
LIN {X 0,Y 446.985,Z 351.858,A -85,B 0,C 180,E1 -8631.525,E2 -8631.525} C_VEL
LIN {X 0,Y 446.73,Z 361.333,A -85,B 0,C 180,E1 -8632.362,E2 -8632.362} C_VEL
LIN {X 0,Y 446.425,Z 368.859,A -85,B 0,C 180,E1 -8633.22,E2 -8633.22} C_VEL
LIN {X 0,Y 446.379,Z 375.101,A -85,B 0,C 180,E1 -8634.127,E2 -8634.127} C_VEL
LIN {X 0,Y 446.174,Z 381.184,A -85,B 0,C 180,E1 -8635.258,E2 -8635.258} C_VEL
LIN {X 0,Y 445.959,Z 385.732,A -85,B 0,C 180,E1 -8636.387,E2 -8636.387} C_VEL
LIN {X 0,Y 445.753,Z 388.448,A -85,B 0,C 180,E1 -8637.29,E2 -8637.29} C_VEL
LIN {X 0,Y 445.61,Z 390.418,A -85,B 0,C 180,E1 -8638.194,E2 -8638.194} C_VEL
LIN {X 0,Y 445.585,Z 391.679,A -85,B 0,C 180,E1 -8639.097,E2 -8639.097} C_VEL
LIN {X 0,Y 445.596,Z 392.263,A -85,B 0,C 180,E1 -8640.001,E2 -8640.001} C_VEL
LIN {X 0,Y 445.622,Z 392.178,A -85,B 0,C 180,E1 -8640.905,E2 -8640.905} C_VEL
LIN {X 0,Y 445.677,Z 391.428,A -85,B 0,C 180,E1 -8641.808,E2 -8641.808} C_VEL
LIN {X 0,Y 445.79,Z 389.995,A -85,B 0,C 180,E1 -8642.712,E2 -8642.712} C_VEL
LIN {X 0,Y 446.016,Z 387.842,A -85,B 0,C 180,E1 -8643.615,E2 -8643.615} C_VEL
LIN {X 0,Y 446.234,Z 384.924,A -85,B 0,C 180,E1 -8644.518,E2 -8644.518} C_VEL
LIN {X 0,Y 446.572,Z 380.052,A -85,B 0,C 180,E1 -8645.646,E2 -8645.646} C_VEL
LIN {X 0,Y 446.823,Z 373.588,A -85,B 0,C 180,E1 -8646.776,E2 -8646.776} C_VEL
LIN {X 0,Y 447.136,Z 366.907,A -85,B 0,C 180,E1 -8647.678,E2 -8647.678} C_VEL
LIN {X 0,Y 447.602,Z 358.41,A -85,B 0,C 180,E1 -8648.579,E2 -8648.579} C_VEL
LIN {X 0,Y 447.968,Z 348.65,A -85,B 0,C 180,E1 -8649.369,E2 -8649.369} C_VEL
LIN {X 0,Y 447.876,Z 343.438,A -85,B 0,C 180,E1 -8649.713,E2 -8649.713} C_VEL
LIN {X 0,Y 445.999,Z 333.925,A -85,B 0,C 180,E1 -8650.298,E2 -8650.298} C_VEL
LIN {X 0,Y 446.167,Z 329.087,A -85,B 0,C 180,E1 -8652.741,E2 -8652.741} C_VEL
LIN {X 0,Y 446.419,Z 321.861,A -85,B 0,C 180,E1 -8656.463,E2 -8656.463} C_VEL
LIN {X 0,Y 446.618,Z 316.518,A -85,B 0,C 180,E1 -8659.298,E2 -8659.298} C_VEL
LIN {X 0,Y 446.854,Z 311.235,A -85,B 0,C 180,E1 -8662.178,E2 -8662.178} C_VEL
LIN {X 0,Y 447.19,Z 306.072,A -85,B 0,C 180,E1 -8665.109,E2 -8665.109} C_VEL
LIN {X 0,Y 447.611,Z 300.32,A -85,B 0,C 180,E1 -8668.446,E2 -8668.446} C_VEL
LIN {X 0,Y 447.713,Z 297.361,A -85,B 0,C 180,E1 -8670.303,E2 -8670.303} C_VEL
LIN {X 0,Y 447.455,Z 294.482,A -85,B 0,C 180,E1 -8672.279,E2 -8672.279} C_VEL
LIN {X 0,Y 446.981,Z 291.582,A -85,B 0,C 180,E1 -8674.475,E2 -8674.475} C_VEL
LIN {X 0,Y 446.418,Z 288.88,A -85,B 0,C 180,E1 -8677.027,E2 -8677.027} C_VEL
LIN {X 0,Y 446.449,Z 288.876,A -85,B 0,C 180,E1 -8680.198,E2 -8680.198} C_VEL
LIN {X 0,Y 446.434,Z 288.878,A -85,B 0,C 180,E1 -8682.605,E2 -8682.605} C_VEL
LIN {X 0,Y 446.457,Z 288.874,A -85,B 0,C 180,E1 -8685.104,E2 -8685.104} C_VEL
LIN {X 0,Y 446.433,Z 288.878,A -85,B 0,C 180,E1 -8688.609,E2 -8688.609} C_VEL
LIN {X 0,Y 446.449,Z 288.888,A -85,B 0,C 180,E1 -8690.973,E2 -8690.973} C_VEL
LIN {X 0,Y 447.583,Z 293.545,A -85,B 0,C 180,E1 -8693.926,E2 -8693.926} C_VEL
LIN {X 0,Y 448.709,Z 298.103,A -85,B 0,C 180,E1 -8696.113,E2 -8696.113} C_VEL
LIN {X 0,Y 450.057,Z 304.038,A -85,B 0,C 180,E1 -8698.457,E2 -8698.457} C_VEL
LIN {X 0,Y 451.214,Z 310.784,A -85,B 0,C 180,E1 -8700.722,E2 -8700.722} C_VEL
LIN {X 0,Y 450.402,Z 317.411,A -85,B 0,C 180,E1 -8702.547,E2 -8702.547} C_VEL
LIN {X 0,Y 448.795,Z 330.924,A -85,B 0,C 180,E1 -8705.974,E2 -8705.974} C_VEL
LIN {X 0,Y 447.817,Z 343.065,A -85,B 0,C 180,E1 -8708.841,E2 -8708.841} C_VEL
LIN {X 0,Y 446.906,Z 357.897,A -85,B 0,C 180,E1 -8712.142,E2 -8712.142} C_VEL
LIN {X 0,Y 446.497,Z 367.677,A -85,B 0,C 180,E1 -8714.244,E2 -8714.244} C_VEL
LIN {X 0,Y 447.903,Z 380.542,A -85,B 0,C 180,E1 -8714.646,E2 -8714.646} C_VEL
LIN {X 0,Y 448.531,Z 391.014,A -85,B 0,C 180,E1 -8715.075,E2 -8715.075} C_VEL
LIN {X 0,Y 448.083,Z 403.089,A -85,B 0,C 180,E1 -8715.698,E2 -8715.698} C_VEL
LIN {X 0,Y 447.519,Z 414.609,A -85,B 0,C 180,E1 -8716.475,E2 -8716.475} C_VEL
LIN {X 0,Y 447.13,Z 425.377,A -85,B 0,C 180,E1 -8717.403,E2 -8717.403} C_VEL
LIN {X 0,Y 446.513,Z 435.043,A -85,B 0,C 180,E1 -8718.423,E2 -8718.423} C_VEL
LIN {X 0,Y 446.165,Z 443.872,A -85,B 0,C 180,E1 -8719.563,E2 -8719.563} C_VEL
LIN {X 0,Y 445.899,Z 452.421,A -85,B 0,C 180,E1 -8720.932,E2 -8720.932} C_VEL
LIN {X 0,Y 445.706,Z 459.294,A -85,B 0,C 180,E1 -8722.297,E2 -8722.297} C_VEL
LIN {X 0,Y 445.601,Z 464.763,A -85,B 0,C 180,E1 -8723.661,E2 -8723.661} C_VEL
LIN {X 0,Y 445.534,Z 469.003,A -85,B 0,C 180,E1 -8725.023,E2 -8725.023} C_VEL
LIN {X 0,Y 445.631,Z 472.145,A -85,B 0,C 180,E1 -8726.383,E2 -8726.383} C_VEL
LIN {X 0,Y 445.662,Z 473.652,A -85,B 0,C 180,E1 -8727.288,E2 -8727.288} C_VEL
LIN {X 0,Y 445.542,Z 474.71,A -85,B 0,C 180,E1 -8728.192,E2 -8728.192} C_VEL
LIN {X 0,Y 445.483,Z 475.367,A -85,B 0,C 180,E1 -8729.096,E2 -8729.096} C_VEL
LIN {X 0,Y 445.486,Z 475.6,A -85,B 0,C 180,E1 -8730,E2 -8730} C_VEL
LIN {X 0,Y 445.539,Z 474.765,A -85,B 0,C 180,E1 -8731.808,E2 -8731.808} C_VEL
LIN {X 0,Y 445.658,Z 473.743,A -85,B 0,C 180,E1 -8732.712,E2 -8732.712} C_VEL
LIN {X 0,Y 445.612,Z 472.224,A -85,B 0,C 180,E1 -8733.617,E2 -8733.617} C_VEL
LIN {X 0,Y 445.526,Z 469.107,A -85,B 0,C 180,E1 -8734.977,E2 -8734.977} C_VEL
LIN {X 0,Y 445.63,Z 464.316,A -85,B 0,C 180,E1 -8736.497,E2 -8736.497} C_VEL
LIN {X 0,Y 445.728,Z 458.389,A -85,B 0,C 180,E1 -8737.93,E2 -8737.93} C_VEL
LIN {X 0,Y 445.926,Z 451.194,A -85,B 0,C 180,E1 -8739.297,E2 -8739.297} C_VEL
LIN {X 0,Y 446.275,Z 442.184,A -85,B 0,C 180,E1 -8740.664,E2 -8740.664} C_VEL
LIN {X 0,Y 446.602,Z 432.851,A -85,B 0,C 180,E1 -8741.805,E2 -8741.805} C_VEL
LIN {X 0,Y 447.143,Z 423.732,A -85,B 0,C 180,E1 -8742.712,E2 -8742.712} C_VEL
LIN {X 0,Y 447.56,Z 412.399,A -85,B 0,C 180,E1 -8743.624,E2 -8743.624} C_VEL
LIN {X 0,Y 448.054,Z 400.666,A -85,B 0,C 180,E1 -8744.361,E2 -8744.361} C_VEL
LIN {X 0,Y 448.384,Z 388.071,A -85,B 0,C 180,E1 -8744.945,E2 -8744.945} C_VEL
LIN {X 0,Y 447.07,Z 374.325,A -85,B 0,C 180,E1 -8745.413,E2 -8745.413} C_VEL
LIN {X 0,Y 446.437,Z 368.566,A -85,B 0,C 180,E1 -8745.57,E2 -8745.57} C_VEL
LIN {X 0,Y 447.087,Z 354.629,A -85,B 0,C 180,E1 -8748.561,E2 -8748.561} C_VEL
LIN {X 0,Y 448.072,Z 337.639,A -85,B 0,C 180,E1 -8752.268,E2 -8752.268} C_VEL
LIN {X 0,Y 449.094,Z 323.196,A -85,B 0,C 180,E1 -8755.49,E2 -8755.49} C_VEL
LIN {X 0,Y 450.266,Z 309.167,A -85,B 0,C 180,E1 -8758.683,E2 -8758.683} C_VEL
LIN {X 0,Y 450.074,Z 305.872,A -85,B 0,C 180,E1 -8759.476,E2 -8759.476} C_VEL
LIN {X 0,Y 447.741,Z 295.046,A -85,B 0,C 180,E1 -8762.255,E2 -8762.255} C_VEL
LIN {X 0,Y 446.449,Z 288.876,A -85,B 0,C 180,E1 -8763.907,E2 -8763.907} C_VEL
LIN {X 0,Y 446.407,Z 288.881,A -85,B 0,C 180,E1 -8766.745,E2 -8766.745} C_VEL
LIN {X 0,Y 446.449,Z 288.875,A -85,B 0,C 180,E1 -8770.198,E2 -8770.198} C_VEL
LIN {X 0,Y 446.435,Z 288.878,A -85,B 0,C 180,E1 -8772.604,E2 -8772.604} C_VEL
LIN {X 0,Y 446.459,Z 288.873,A -85,B 0,C 180,E1 -8775.103,E2 -8775.103} C_VEL
LIN {X 0,Y 446.433,Z 288.876,A -85,B 0,C 180,E1 -8778.609,E2 -8778.609} C_VEL
LIN {X 0,Y 446.461,Z 288.874,A -85,B 0,C 180,E1 -8780.974,E2 -8780.974} C_VEL
LIN {X 0,Y 446.423,Z 288.88,A -85,B 0,C 180,E1 -8784.373,E2 -8784.373} C_VEL
LIN {X 0,Y 446.425,Z 288.883,A -85,B 0,C 180,E1 -8787.638,E2 -8787.638} C_VEL
LIN {X 0,Y 446.373,Z 288.985,A -85,B 0,C 180,E1 -8790.849,E2 -8790.849} C_VEL
LIN {X 0,Y 446.534,Z 293,A -85,B 0,C 180,E1 -8792.334,E2 -8792.334} C_VEL
LIN {X 0,Y 446.483,Z 300.909,A -85,B 0,C 180,E1 -8795.345,E2 -8795.345} C_VEL
LIN {X 0,Y 446.416,Z 308.125,A -85,B 0,C 180,E1 -8798.256,E2 -8798.256} C_VEL
LIN {X 0,Y 446.398,Z 314.598,A -85,B 0,C 180,E1 -8800.845,E2 -8800.845} C_VEL
LIN {X 0,Y 446.321,Z 321.787,A -85,B 0,C 180,E1 -8803.851,E2 -8803.851} C_VEL
LIN {X 0,Y 446.298,Z 329.81,A -85,B 0,C 180,E1 -8807.263,E2 -8807.263} C_VEL
LIN {X 0,Y 446.275,Z 336.218,A -85,B 0,C 180,E1 -8810.023,E2 -8810.023} C_VEL
LIN {X 0,Y 446.248,Z 337.496,A -85,B 0,C 180,E1 -8810.566,E2 -8810.566} C_VEL
LIN {X 0,Y 447.373,Z 344.167,A -85,B 0,C 180,E1 -8810.904,E2 -8810.904} C_VEL
LIN {X 0,Y 447.213,Z 352.557,A -85,B 0,C 180,E1 -8811.413,E2 -8811.413} C_VEL
LIN {X 0,Y 447.005,Z 361.161,A -85,B 0,C 180,E1 -8812.103,E2 -8812.103} C_VEL
LIN {X 0,Y 446.665,Z 367.513,A -85,B 0,C 180,E1 -8812.768,E2 -8812.768} C_VEL
LIN {X 0,Y 446.544,Z 374.353,A -85,B 0,C 180,E1 -8813.674,E2 -8813.674} C_VEL
LIN {X 0,Y 446.326,Z 379.652,A -85,B 0,C 180,E1 -8814.578,E2 -8814.578} C_VEL
LIN {X 0,Y 446.224,Z 383.764,A -85,B 0,C 180,E1 -8815.482,E2 -8815.482} C_VEL
LIN {X 0,Y 446.263,Z 385.509,A -85,B 0,C 180,E1 -8815.935,E2 -8815.935} C_VEL
LIN {X 0,Y 446.033,Z 388.261,A -85,B 0,C 180,E1 -8816.837,E2 -8816.837} C_VEL
LIN {X 0,Y 445.763,Z 389.363,A -85,B 0,C 180,E1 -8817.288,E2 -8817.288} C_VEL
LIN {X 0,Y 445.652,Z 390.988,A -85,B 0,C 180,E1 -8818.191,E2 -8818.191} C_VEL
LIN {X 0,Y 445.6,Z 391.892,A -85,B 0,C 180,E1 -8819.095,E2 -8819.095} C_VEL
LIN {X 0,Y 445.574,Z 392.104,A -85,B 0,C 180,E1 -8819.999,E2 -8819.999} C_VEL
LIN {X 0,Y 445.566,Z 391.63,A -85,B 0,C 180,E1 -8820.903,E2 -8820.903} C_VEL
LIN {X 0,Y 445.603,Z 390.459,A -85,B 0,C 180,E1 -8821.806,E2 -8821.806} C_VEL
LIN {X 0,Y 445.923,Z 387.376,A -85,B 0,C 180,E1 -8823.161,E2 -8823.161} C_VEL
LIN {X 0,Y 446.032,Z 384.328,A -85,B 0,C 180,E1 -8824.065,E2 -8824.065} C_VEL
LIN {X 0,Y 446.207,Z 379.165,A -85,B 0,C 180,E1 -8825.195,E2 -8825.195} C_VEL
LIN {X 0,Y 446.371,Z 373.843,A -85,B 0,C 180,E1 -8826.1,E2 -8826.1} C_VEL
LIN {X 0,Y 446.413,Z 367.238,A -85,B 0,C 180,E1 -8826.969,E2 -8826.969} C_VEL
LIN {X 0,Y 446.655,Z 359.591,A -85,B 0,C 180,E1 -8827.764,E2 -8827.764} C_VEL
LIN {X 0,Y 446.822,Z 350.356,A -85,B 0,C 180,E1 -8828.478,E2 -8828.478} C_VEL
LIN {X 0,Y 446.83,Z 341.443,A -85,B 0,C 180,E1 -8828.991,E2 -8828.991} C_VEL
LIN {X 0,Y 445.928,Z 335.587,A -85,B 0,C 180,E1 -8829.267,E2 -8829.267} C_VEL
LIN {X 0,Y 446.036,Z 327.435,A -85,B 0,C 180,E1 -8832.742,E2 -8832.742} C_VEL
LIN {X 0,Y 446.057,Z 318.784,A -85,B 0,C 180,E1 -8836.474,E2 -8836.474} C_VEL
LIN {X 0,Y 446.135,Z 311.1,A -85,B 0,C 180,E1 -8839.796,E2 -8839.796} C_VEL
LIN {X 0,Y 446.176,Z 303.261,A -85,B 0,C 180,E1 -8843.189,E2 -8843.189} C_VEL
LIN {X 0,Y 446.27,Z 296.351,A -85,B 0,C 180,E1 -8846.163,E2 -8846.163} C_VEL
LIN {X 0,Y 446.441,Z 288.877,A -85,B 0,C 180,E1 -8849.46,E2 -8849.46} C_VEL
LIN {X 0,Y 446.403,Z 288.875,A -85,B 0,C 180,E1 -8852.361,E2 -8852.361} C_VEL
LIN {X 0,Y 446.41,Z 288.877,A -85,B 0,C 180,E1 -8855.625,E2 -8855.625} C_VEL
LIN {X 0,Y 446.414,Z 288.881,A -85,B 0,C 180,E1 -8859.028,E2 -8859.028} C_VEL
LIN {X 0,Y 446.412,Z 288.877,A -85,B 0,C 180,E1 -8862.274,E2 -8862.274} C_VEL
LIN {X 0,Y 446.443,Z 288.874,A -85,B 0,C 180,E1 -8865.103,E2 -8865.103} C_VEL
LIN {X 0,Y 446.42,Z 288.88,A -85,B 0,C 180,E1 -8868.608,E2 -8868.608} C_VEL
LIN {X 0,Y 446.452,Z 288.872,A -85,B 0,C 180,E1 -8870.974,E2 -8870.974} C_VEL
LIN {X 0,Y 446.412,Z 288.88,A -85,B 0,C 180,E1 -8874.373,E2 -8874.373} C_VEL
LIN {X 0,Y 446.42,Z 288.877,A -85,B 0,C 180,E1 -8877.638,E2 -8877.638} C_VEL
LIN {X 0,Y 446.46,Z 288.871,A -85,B 0,C 180,E1 -8880.791,E2 -8880.791} C_VEL
LIN {X 0,Y 446.467,Z 288.872,A -85,B 0,C 180,E1 -8883.848,E2 -8883.848} C_VEL
LIN {X 0,Y 446.418,Z 288.878,A -85,B 0,C 180,E1 -8886.823,E2 -8886.823} C_VEL
LIN {X 0,Y 446.434,Z 288.876,A -85,B 0,C 180,E1 -8889.737,E2 -8889.737} C_VEL
LIN {X 0,Y 446.452,Z 288.875,A -85,B 0,C 180,E1 -8892.597,E2 -8892.597} C_VEL
LIN {X 0,Y 446.458,Z 288.872,A -85,B 0,C 180,E1 -8895.412,E2 -8895.412} C_VEL
LIN {X 0,Y 446.504,Z 288.867,A -85,B 0,C 180,E1 -8898.193,E2 -8898.193} C_VEL
LIN {X 0,Y 446.52,Z 288.863,A -85,B 0,C 180,E1 -8900.944,E2 -8900.944} C_VEL
LIN {X 0,Y 446.603,Z 288.852,A -85,B 0,C 180,E1 -8903.676,E2 -8903.676} C_VEL
LIN {X 0,Y 446.415,Z 288.876,A -85,B 0,C 180,E1 -8906.158,E2 -8906.158} C_VEL
LIN {X 0,Y 445.817,Z 288.956,A -85,B 0,C 180,E1 -8906.911,E2 -8906.911} C_VEL
LIN {X 0,Y 443.167,Z 289.293,A -85,B 0,C 180,E1 -8908.138,E2 -8908.138} C_VEL
LIN {X 0,Y 440.031,Z 289.68,A -85,B 0,C 180,E1 -8909.633,E2 -8909.633} C_VEL
LIN {X 0,Y 439.636,Z 289.723,A -85,B 0,C 180,E1 -8910.147,E2 -8910.147} C_VEL
LIN {X 0,Y 439.595,Z 289.724,A -85,B 0,C 180,E1 -8912.749,E2 -8912.749} C_VEL
LIN {X 0,Y 439.554,Z 289.73,A -85,B 0,C 180,E1 -8916.426,E2 -8916.426} C_VEL
LIN {X 0,Y 439.483,Z 289.741,A -85,B 0,C 180,E1 -8919.202,E2 -8919.202} C_VEL
LIN {X 0,Y 439.453,Z 289.744,A -85,B 0,C 180,E1 -8922.938,E2 -8922.938} C_VEL
LIN {X 0,Y 439.435,Z 289.747,A -85,B 0,C 180,E1 -8926.349,E2 -8926.349} C_VEL
LIN {X 0,Y 439.391,Z 289.752,A -85,B 0,C 180,E1 -8929.627,E2 -8929.627} C_VEL
LIN {X 0,Y 439.354,Z 289.757,A -85,B 0,C 180,E1 -8932.576,E2 -8932.576} C_VEL
LIN {X 0,Y 439.395,Z 289.752,A -85,B 0,C 180,E1 -8935.586,E2 -8935.586} C_VEL
LIN {X 0,Y 439.415,Z 289.75,A -85,B 0,C 180,E1 -8938.674,E2 -8938.674} C_VEL
LIN {X 0,Y 439.373,Z 289.755,A -85,B 0,C 180,E1 -8942.034,E2 -8942.034} C_VEL
LIN {X 0,Y 439.387,Z 289.753,A -85,B 0,C 180,E1 -8945.342,E2 -8945.342} C_VEL
LIN {X 0,Y 439.382,Z 289.753,A -85,B 0,C 180,E1 -8948.595,E2 -8948.595} C_VEL
LIN {X 0,Y 439.38,Z 289.756,A -85,B 0,C 180,E1 -8951.258,E2 -8951.258} C_VEL
LIN {X 0,Y 439.391,Z 289.752,A -85,B 0,C 180,E1 -8954.731,E2 -8954.731} C_VEL
LIN {X 0,Y 439.375,Z 289.753,A -85,B 0,C 180,E1 -8957.795,E2 -8957.795} C_VEL
LIN {X 0,Y 439.355,Z 289.756,A -85,B 0,C 180,E1 -8961.404,E2 -8961.404} C_VEL
LIN {X 0,Y 439.388,Z 289.756,A -85,B 0,C 180,E1 -8964.845,E2 -8964.845} C_VEL
LIN {X 0,Y 439.422,Z 289.747,A -85,B 0,C 180,E1 -8968.145,E2 -8968.145} C_VEL
LIN {X 0,Y 439.502,Z 289.953,A -85,B 0,C 180,E1 -8969.5,E2 -8969.5} C_VEL
LIN {X 0,Y 439.498,Z 293.96,A -85,B 0,C 180,E1 -8971.583,E2 -8971.583} C_VEL
LIN {X 0,Y 439.254,Z 299.498,A -85,B 0,C 180,E1 -8974.407,E2 -8974.407} C_VEL
LIN {X 0,Y 439.075,Z 305.437,A -85,B 0,C 180,E1 -8977.41,E2 -8977.41} C_VEL
LIN {X 0,Y 438.967,Z 312.34,A -85,B 0,C 180,E1 -8980.841,E2 -8980.841} C_VEL
LIN {X 0,Y 438.786,Z 319.205,A -85,B 0,C 180,E1 -8984.201,E2 -8984.201} C_VEL
LIN {X 0,Y 438.723,Z 327.059,A -85,B 0,C 180,E1 -8987.982,E2 -8987.982} C_VEL
LIN {X 0,Y 438.569,Z 331.745,A -85,B 0,C 180,E1 -8990.198,E2 -8990.198} C_VEL
LIN {X 0,Y 440.12,Z 342.597,A -85,B 0,C 180,E1 -8990.755,E2 -8990.755} C_VEL
LIN {X 0,Y 439.977,Z 352.049,A -85,B 0,C 180,E1 -8991.389,E2 -8991.389} C_VEL
LIN {X 0,Y 439.724,Z 361.596,A -85,B 0,C 180,E1 -8992.24,E2 -8992.24} C_VEL
LIN {X 0,Y 439.4,Z 369.243,A -85,B 0,C 180,E1 -8993.121,E2 -8993.121} C_VEL
LIN {X 0,Y 439.291,Z 376.848,A -85,B 0,C 180,E1 -8994.263,E2 -8994.263} C_VEL
LIN {X 0,Y 439.079,Z 382.668,A -85,B 0,C 180,E1 -8995.411,E2 -8995.411} C_VEL
LIN {X 0,Y 438.866,Z 387.717,A -85,B 0,C 180,E1 -8996.788,E2 -8996.788} C_VEL
LIN {X 0,Y 438.551,Z 391.02,A -85,B 0,C 180,E1 -8998.165,E2 -8998.165} C_VEL
LIN {X 0,Y 438.516,Z 392.323,A -85,B 0,C 180,E1 -8999.083,E2 -8999.083} C_VEL
LIN {X 0,Y 438.53,Z 392.946,A -85,B 0,C 180,E1 -9000.001,E2 -9000.001} C_VEL
LIN {X 0,Y 438.56,Z 392.899,A -85,B 0,C 180,E1 -9000.919,E2 -9000.919} C_VEL
LIN {X 0,Y 438.621,Z 392.184,A -85,B 0,C 180,E1 -9001.838,E2 -9001.838} C_VEL
LIN {X 0,Y 438.744,Z 390.787,A -85,B 0,C 180,E1 -9002.756,E2 -9002.756} C_VEL
LIN {X 0,Y 438.983,Z 388.67,A -85,B 0,C 180,E1 -9003.673,E2 -9003.673} C_VEL
LIN {X 0,Y 439.214,Z 385.809,A -85,B 0,C 180,E1 -9004.59,E2 -9004.59} C_VEL
LIN {X 0,Y 439.57,Z 381.027,A -85,B 0,C 180,E1 -9005.736,E2 -9005.736} C_VEL
LIN {X 0,Y 439.875,Z 374.694,A -85,B 0,C 180,E1 -9006.883,E2 -9006.883} C_VEL
LIN {X 0,Y 440.228,Z 367.845,A -85,B 0,C 180,E1 -9007.841,E2 -9007.841} C_VEL
LIN {X 0,Y 440.701,Z 359.863,A -85,B 0,C 180,E1 -9008.714,E2 -9008.714} C_VEL
LIN {X 0,Y 441.105,Z 350.421,A -85,B 0,C 180,E1 -9009.516,E2 -9009.516} C_VEL
LIN {X 0,Y 441.129,Z 345.421,A -85,B 0,C 180,E1 -9009.863,E2 -9009.863} C_VEL
LIN {X 0,Y 439.5,Z 336.702,A -85,B 0,C 180,E1 -9010.423,E2 -9010.423} C_VEL
LIN {X 0,Y 438.98,Z 334.439,A -85,B 0,C 180,E1 -9010.552,E2 -9010.552} C_VEL
LIN {X 0,Y 439.15,Z 329.77,A -85,B 0,C 180,E1 -9012.948,E2 -9012.948} C_VEL
LIN {X 0,Y 439.427,Z 323.29,A -85,B 0,C 180,E1 -9016.338,E2 -9016.338} C_VEL
LIN {X 0,Y 439.662,Z 317.22,A -85,B 0,C 180,E1 -9019.615,E2 -9019.615} C_VEL
LIN {X 0,Y 439.931,Z 312.052,A -85,B 0,C 180,E1 -9022.546,E2 -9022.546} C_VEL
LIN {X 0,Y 440.27,Z 306.815,A -85,B 0,C 180,E1 -9025.532,E2 -9025.532} C_VEL
LIN {X 0,Y 440.725,Z 301.571,A -85,B 0,C 180,E1 -9028.71,E2 -9028.71} C_VEL
LIN {X 0,Y 440.788,Z 298.565,A -85,B 0,C 180,E1 -9030.679,E2 -9030.679} C_VEL
LIN {X 0,Y 440.51,Z 295.586,A -85,B 0,C 180,E1 -9032.851,E2 -9032.851} C_VEL
LIN {X 0,Y 439.969,Z 292.462,A -85,B 0,C 180,E1 -9035.445,E2 -9035.445} C_VEL
LIN {X 0,Y 439.38,Z 289.757,A -85,B 0,C 180,E1 -9038.393,E2 -9038.393} C_VEL
LIN {X 0,Y 439.394,Z 289.754,A -85,B 0,C 180,E1 -9041.257,E2 -9041.257} C_VEL
LIN {X 0,Y 439.405,Z 289.753,A -85,B 0,C 180,E1 -9044.73,E2 -9044.73} C_VEL
LIN {X 0,Y 439.401,Z 289.754,A -85,B 0,C 180,E1 -9047.796,E2 -9047.796} C_VEL
LIN {X 0,Y 439.423,Z 289.825,A -85,B 0,C 180,E1 -9049.477,E2 -9049.477} C_VEL
LIN {X 0,Y 439.998,Z 292.251,A -85,B 0,C 180,E1 -9051.507,E2 -9051.507} C_VEL
LIN {X 0,Y 441.142,Z 296.869,A -85,B 0,C 180,E1 -9054.342,E2 -9054.342} C_VEL
LIN {X 0,Y 442.422,Z 302.078,A -85,B 0,C 180,E1 -9056.768,E2 -9056.768} C_VEL
LIN {X 0,Y 443.732,Z 308.375,A -85,B 0,C 180,E1 -9059.195,E2 -9059.195} C_VEL
LIN {X 0,Y 444.406,Z 312.686,A -85,B 0,C 180,E1 -9060.643,E2 -9060.643} C_VEL
LIN {X 0,Y 443.443,Z 319.793,A -85,B 0,C 180,E1 -9062.638,E2 -9062.638} C_VEL
LIN {X 0,Y 442.017,Z 331.151,A -85,B 0,C 180,E1 -9065.582,E2 -9065.582} C_VEL
LIN {X 0,Y 440.853,Z 344.072,A -85,B 0,C 180,E1 -9068.735,E2 -9068.735} C_VEL
LIN {X 0,Y 439.885,Z 358.764,A -85,B 0,C 180,E1 -9072.088,E2 -9072.088} C_VEL
LIN {X 0,Y 439.474,Z 367.434,A -85,B 0,C 180,E1 -9073.991,E2 -9073.991} C_VEL
LIN {X 0,Y 440.939,Z 379.457,A -85,B 0,C 180,E1 -9074.368,E2 -9074.368} C_VEL
LIN {X 0,Y 441.618,Z 391.865,A -85,B 0,C 180,E1 -9074.895,E2 -9074.895} C_VEL
LIN {X 0,Y 441.085,Z 404.49,A -85,B 0,C 180,E1 -9075.584,E2 -9075.584} C_VEL
LIN {X 0,Y 440.497,Z 415.606,A -85,B 0,C 180,E1 -9076.381,E2 -9076.381} C_VEL
LIN {X 0,Y 440.043,Z 427.166,A -85,B 0,C 180,E1 -9077.431,E2 -9077.431} C_VEL
LIN {X 0,Y 439.442,Z 436.36,A -85,B 0,C 180,E1 -9078.468,E2 -9078.468} C_VEL
LIN {X 0,Y 439.072,Z 444.797,A -85,B 0,C 180,E1 -9079.626,E2 -9079.626} C_VEL
LIN {X 0,Y 438.78,Z 453.067,A -85,B 0,C 180,E1 -9081.015,E2 -9081.015} C_VEL
LIN {X 0,Y 438.614,Z 458.661,A -85,B 0,C 180,E1 -9082.172,E2 -9082.172} C_VEL
LIN {X 0,Y 438.548,Z 464.127,A -85,B 0,C 180,E1 -9083.559,E2 -9083.559} C_VEL
LIN {X 0,Y 438.471,Z 468.363,A -85,B 0,C 180,E1 -9084.942,E2 -9084.942} C_VEL
LIN {X 0,Y 438.562,Z 471.501,A -85,B 0,C 180,E1 -9086.325,E2 -9086.325} C_VEL
LIN {X 0,Y 438.592,Z 472.999,A -85,B 0,C 180,E1 -9087.245,E2 -9087.245} C_VEL
LIN {X 0,Y 438.486,Z 474.054,A -85,B 0,C 180,E1 -9088.163,E2 -9088.163} C_VEL
LIN {X 0,Y 438.42,Z 474.706,A -85,B 0,C 180,E1 -9089.081,E2 -9089.081} C_VEL
LIN {X 0,Y 438.419,Z 474.924,A -85,B 0,C 180,E1 -9090,E2 -9090} C_VEL
LIN {X 0,Y 438.417,Z 474.699,A -85,B 0,C 180,E1 -9090.919,E2 -9090.919} C_VEL
LIN {X 0,Y 438.483,Z 474.076,A -85,B 0,C 180,E1 -9091.837,E2 -9091.837} C_VEL
LIN {X 0,Y 438.604,Z 473.038,A -85,B 0,C 180,E1 -9092.755,E2 -9092.755} C_VEL
LIN {X 0,Y 438.543,Z 471.5,A -85,B 0,C 180,E1 -9093.675,E2 -9093.675} C_VEL
LIN {X 0,Y 438.464,Z 468.354,A -85,B 0,C 180,E1 -9095.058,E2 -9095.058} C_VEL
LIN {X 0,Y 438.549,Z 463.927,A -85,B 0,C 180,E1 -9096.488,E2 -9096.488} C_VEL
LIN {X 0,Y 438.669,Z 457.544,A -85,B 0,C 180,E1 -9098.059,E2 -9098.059} C_VEL
LIN {X 0,Y 438.854,Z 450.267,A -85,B 0,C 180,E1 -9099.448,E2 -9099.448} C_VEL
LIN {X 0,Y 439.24,Z 441.184,A -85,B 0,C 180,E1 -9100.836,E2 -9100.836} C_VEL
LIN {X 0,Y 439.631,Z 431.71,A -85,B 0,C 180,E1 -9101.995,E2 -9101.995} C_VEL
LIN {X 0,Y 440.09,Z 423.749,A -85,B 0,C 180,E1 -9102.802,E2 -9102.802} C_VEL
LIN {X 0,Y 440.515,Z 412.685,A -85,B 0,C 180,E1 -9103.717,E2 -9103.717} C_VEL
LIN {X 0,Y 440.949,Z 401.931,A -85,B 0,C 180,E1 -9104.421,E2 -9104.421} C_VEL
LIN {X 0,Y 441.379,Z 390.488,A -85,B 0,C 180,E1 -9104.996,E2 -9104.996} C_VEL
LIN {X 0,Y 440.414,Z 377.848,A -85,B 0,C 180,E1 -9105.474,E2 -9105.474} C_VEL
LIN {X 0,Y 439.403,Z 368.304,A -85,B 0,C 180,E1 -9105.748,E2 -9105.748} C_VEL
LIN {X 0,Y 440.036,Z 355.176,A -85,B 0,C 180,E1 -9108.628,E2 -9108.628} C_VEL
LIN {X 0,Y 441.078,Z 338.523,A -85,B 0,C 180,E1 -9112.342,E2 -9112.342} C_VEL
LIN {X 0,Y 442.27,Z 322.802,A -85,B 0,C 180,E1 -9115.912,E2 -9115.912} C_VEL
LIN {X 0,Y 443.368,Z 310.176,A -85,B 0,C 180,E1 -9118.85,E2 -9118.85} C_VEL
LIN {X 0,Y 442.786,Z 305.597,A -85,B 0,C 180,E1 -9119.999,E2 -9119.999} C_VEL
LIN {X 0,Y 440.46,Z 294.716,A -85,B 0,C 180,E1 -9122.855,E2 -9122.855} C_VEL
LIN {X 0,Y 439.41,Z 289.753,A -85,B 0,C 180,E1 -9124.25,E2 -9124.25} C_VEL
LIN {X 0,Y 439.353,Z 289.76,A -85,B 0,C 180,E1 -9127.435,E2 -9127.435} C_VEL
LIN {X 0,Y 439.407,Z 289.752,A -85,B 0,C 180,E1 -9129.849,E2 -9129.849} C_VEL
LIN {X 0,Y 439.387,Z 289.755,A -85,B 0,C 180,E1 -9132.627,E2 -9132.627} C_VEL
LIN {X 0,Y 439.407,Z 289.752,A -85,B 0,C 180,E1 -9135.27,E2 -9135.27} C_VEL
LIN {X 0,Y 439.394,Z 289.754,A -85,B 0,C 180,E1 -9138.743,E2 -9138.743} C_VEL
LIN {X 0,Y 439.382,Z 289.756,A -85,B 0,C 180,E1 -9141.607,E2 -9141.607} C_VEL
LIN {X 0,Y 439.402,Z 289.754,A -85,B 0,C 180,E1 -9144.843,E2 -9144.843} C_VEL
LIN {X 0,Y 439.376,Z 289.761,A -85,B 0,C 180,E1 -9148.139,E2 -9148.139} C_VEL
LIN {X 0,Y 439.385,Z 289.898,A -85,B 0,C 180,E1 -9150.603,E2 -9150.603} C_VEL
LIN {X 0,Y 439.593,Z 294.611,A -85,B 0,C 180,E1 -9152.377,E2 -9152.377} C_VEL
LIN {X 0,Y 439.529,Z 303.236,A -85,B 0,C 180,E1 -9155.703,E2 -9155.703} C_VEL
LIN {X 0,Y 439.438,Z 311.167,A -85,B 0,C 180,E1 -9158.908,E2 -9158.908} C_VEL
LIN {X 0,Y 439.37,Z 318.169,A -85,B 0,C 180,E1 -9161.824,E2 -9161.824} C_VEL
LIN {X 0,Y 439.33,Z 326.139,A -85,B 0,C 180,E1 -9165.169,E2 -9165.169} C_VEL
LIN {X 0,Y 439.358,Z 333.791,A -85,B 0,C 180,E1 -9168.465,E2 -9168.465} C_VEL
LIN {X 0,Y 439.306,Z 338.392,A -85,B 0,C 180,E1 -9170.372,E2 -9170.372} C_VEL
LIN {X 0,Y 440.47,Z 344.733,A -85,B 0,C 180,E1 -9170.702,E2 -9170.702} C_VEL
LIN {X 0,Y 440.271,Z 353.926,A -85,B 0,C 180,E1 -9171.276,E2 -9171.276} C_VEL
LIN {X 0,Y 440.073,Z 362.041,A -85,B 0,C 180,E1 -9171.951,E2 -9171.951} C_VEL
LIN {X 0,Y 439.697,Z 368.559,A -85,B 0,C 180,E1 -9172.652,E2 -9172.652} C_VEL
LIN {X 0,Y 439.558,Z 375.312,A -85,B 0,C 180,E1 -9173.573,E2 -9173.573} C_VEL
LIN {X 0,Y 439.313,Z 380.527,A -85,B 0,C 180,E1 -9174.491,E2 -9174.491} C_VEL
LIN {X 0,Y 439.202,Z 384.605,A -85,B 0,C 180,E1 -9175.41,E2 -9175.41} C_VEL
LIN {X 0,Y 439.238,Z 386.329,A -85,B 0,C 180,E1 -9175.87,E2 -9175.87} C_VEL
LIN {X 0,Y 438.999,Z 389.046,A -85,B 0,C 180,E1 -9176.787,E2 -9176.787} C_VEL
LIN {X 0,Y 438.716,Z 390.148,A -85,B 0,C 180,E1 -9177.244,E2 -9177.244} C_VEL
LIN {X 0,Y 438.596,Z 391.738,A -85,B 0,C 180,E1 -9178.162,E2 -9178.162} C_VEL
LIN {X 0,Y 438.538,Z 392.606,A -85,B 0,C 180,E1 -9179.081,E2 -9179.081} C_VEL
LIN {X 0,Y 438.507,Z 392.78,A -85,B 0,C 180,E1 -9179.999,E2 -9179.999} C_VEL
LIN {X 0,Y 438.497,Z 392.264,A -85,B 0,C 180,E1 -9180.917,E2 -9180.917} C_VEL
LIN {X 0,Y 438.544,Z 391.053,A -85,B 0,C 180,E1 -9181.836,E2 -9181.836} C_VEL
LIN {X 0,Y 438.863,Z 387.912,A -85,B 0,C 180,E1 -9183.212,E2 -9183.212} C_VEL
LIN {X 0,Y 438.967,Z 384.799,A -85,B 0,C 180,E1 -9184.13,E2 -9184.13} C_VEL
LIN {X 0,Y 439.17,Z 379.57,A -85,B 0,C 180,E1 -9185.278,E2 -9185.278} C_VEL
LIN {X 0,Y 439.329,Z 374.158,A -85,B 0,C 180,E1 -9186.198,E2 -9186.198} C_VEL
LIN {X 0,Y 439.396,Z 367.254,A -85,B 0,C 180,E1 -9187.104,E2 -9187.104} C_VEL
LIN {X 0,Y 439.649,Z 359.281,A -85,B 0,C 180,E1 -9187.923,E2 -9187.923} C_VEL
LIN {X 0,Y 439.793,Z 350.259,A -85,B 0,C 180,E1 -9188.615,E2 -9188.615} C_VEL
LIN {X 0,Y 439.814,Z 342.251,A -85,B 0,C 180,E1 -9189.078,E2 -9189.078} C_VEL
LIN {X 0,Y 438.88,Z 336.115,A -85,B 0,C 180,E1 -9189.388,E2 -9189.388} C_VEL
LIN {X 0,Y 439.032,Z 328.932,A -85,B 0,C 180,E1 -9192.449,E2 -9192.449} C_VEL
LIN {X 0,Y 438.992,Z 320.382,A -85,B 0,C 180,E1 -9196.143,E2 -9196.143} C_VEL
LIN {X 0,Y 439.098,Z 312.313,A -85,B 0,C 180,E1 -9199.639,E2 -9199.639} C_VEL
LIN {X 0,Y 439.125,Z 304.389,A -85,B 0,C 180,E1 -9203.084,E2 -9203.084} C_VEL
LIN {X 0,Y 439.24,Z 296.86,A -85,B 0,C 180,E1 -9206.36,E2 -9206.36} C_VEL
LIN {X 0,Y 439.4,Z 289.754,A -85,B 0,C 180,E1 -9209.459,E2 -9209.459} C_VEL
LIN {X 0,Y 439.362,Z 289.756,A -85,B 0,C 180,E1 -9212.945,E2 -9212.945} C_VEL
LIN {X 0,Y 439.365,Z 289.753,A -85,B 0,C 180,E1 -9216.286,E2 -9216.286} C_VEL
LIN {X 0,Y 439.369,Z 289.753,A -85,B 0,C 180,E1 -9219.844,E2 -9219.844} C_VEL
LIN {X 0,Y 439.362,Z 289.757,A -85,B 0,C 180,E1 -9222.624,E2 -9222.624} C_VEL
LIN {X 0,Y 439.391,Z 289.752,A -85,B 0,C 180,E1 -9225.269,E2 -9225.269} C_VEL
LIN {X 0,Y 439.38,Z 289.756,A -85,B 0,C 180,E1 -9228.742,E2 -9228.742} C_VEL
LIN {X 0,Y 439.377,Z 289.754,A -85,B 0,C 180,E1 -9231.605,E2 -9231.605} C_VEL
LIN {X 0,Y 439.392,Z 289.752,A -85,B 0,C 180,E1 -9234.843,E2 -9234.843} C_VEL
LIN {X 0,Y 439.377,Z 289.756,A -85,B 0,C 180,E1 -9238.14,E2 -9238.14} C_VEL
LIN {X 0,Y 439.415,Z 289.75,A -85,B 0,C 180,E1 -9241.326,E2 -9241.326} C_VEL
LIN {X 0,Y 439.395,Z 289.752,A -85,B 0,C 180,E1 -9244.414,E2 -9244.414} C_VEL
LIN {X 0,Y 439.354,Z 289.757,A -85,B 0,C 180,E1 -9247.424,E2 -9247.424} C_VEL
LIN {X 0,Y 439.43,Z 289.749,A -85,B 0,C 180,E1 -9250.662,E2 -9250.662} C_VEL
LIN {X 0,Y 439.45,Z 289.745,A -85,B 0,C 180,E1 -9254.224,E2 -9254.224} C_VEL
LIN {X 0,Y 439.47,Z 289.742,A -85,B 0,C 180,E1 -9258.001,E2 -9258.001} C_VEL
LIN {X 0,Y 439.491,Z 289.738,A -85,B 0,C 180,E1 -9261.725,E2 -9261.725} C_VEL
LIN {X 0,Y 439.594,Z 289.728,A -85,B 0,C 180,E1 -9264.495,E2 -9264.495} C_VEL
LIN {X 0,Y 439.613,Z 289.727,A -85,B 0,C 180,E1 -9268.168,E2 -9268.168} C_VEL
LIN {X 0,Y 439.636,Z 289.723,A -85,B 0,C 180,E1 -9270.147,E2 -9270.147} C_VEL
LIN {X 0,Y 438.821,Z 289.82,A -85,B 0,C 180,E1 -9270.912,E2 -9270.912} C_VEL
LIN {X 0,Y 435.842,Z 290.195,A -85,B 0,C 180,E1 -9272.154,E2 -9272.154} C_VEL
LIN {X 0,Y 433.417,Z 290.498,A -85,B 0,C 180,E1 -9273.156,E2 -9273.156} C_VEL
LIN {X 0,Y 432.407,Z 290.625,A -85,B 0,C 180,E1 -9273.932,E2 -9273.932} C_VEL
LIN {X 0,Y 432.337,Z 290.629,A -85,B 0,C 180,E1 -9274.194,E2 -9274.194} C_VEL
LIN {X 0,Y 432.568,Z 290.604,A -85,B 0,C 180,E1 -9275.594,E2 -9275.594} C_VEL
LIN {X 0,Y 432.451,Z 290.615,A -85,B 0,C 180,E1 -9278.411,E2 -9278.411} C_VEL
LIN {X 0,Y 432.446,Z 290.616,A -85,B 0,C 180,E1 -9282.197,E2 -9282.197} C_VEL
LIN {X 0,Y 432.419,Z 290.62,A -85,B 0,C 180,E1 -9286.039,E2 -9286.039} C_VEL
LIN {X 0,Y 432.376,Z 290.627,A -85,B 0,C 180,E1 -9289.486,E2 -9289.486} C_VEL
LIN {X 0,Y 432.308,Z 290.636,A -85,B 0,C 180,E1 -9292.965,E2 -9292.965} C_VEL
LIN {X 0,Y 432.354,Z 290.63,A -85,B 0,C 180,E1 -9296.033,E2 -9296.033} C_VEL
LIN {X 0,Y 432.343,Z 290.63,A -85,B 0,C 180,E1 -9299.188,E2 -9299.188} C_VEL
LIN {X 0,Y 432.322,Z 290.633,A -85,B 0,C 180,E1 -9302.296,E2 -9302.296} C_VEL
LIN {X 0,Y 432.332,Z 290.632,A -85,B 0,C 180,E1 -9304.678,E2 -9304.678} C_VEL
LIN {X 0,Y 432.339,Z 290.63,A -85,B 0,C 180,E1 -9308.15,E2 -9308.15} C_VEL
LIN {X 0,Y 432.324,Z 290.634,A -85,B 0,C 180,E1 -9311.603,E2 -9311.603} C_VEL
LIN {X 0,Y 432.326,Z 290.631,A -85,B 0,C 180,E1 -9314.349,E2 -9314.349} C_VEL
LIN {X 0,Y 432.309,Z 290.637,A -85,B 0,C 180,E1 -9317.018,E2 -9317.018} C_VEL
LIN {X 0,Y 432.284,Z 290.635,A -85,B 0,C 180,E1 -9319.829,E2 -9319.829} C_VEL
LIN {X 0,Y 432.298,Z 290.638,A -85,B 0,C 180,E1 -9323.023,E2 -9323.023} C_VEL
LIN {X 0,Y 432.327,Z 290.629,A -85,B 0,C 180,E1 -9326.003,E2 -9326.003} C_VEL
LIN {X 0,Y 432.434,Z 290.625,A -85,B 0,C 180,E1 -9329.328,E2 -9329.328} C_VEL
LIN {X 0,Y 432.472,Z 294.43,A -85,B 0,C 180,E1 -9331.348,E2 -9331.348} C_VEL
LIN {X 0,Y 432.21,Z 300.51,A -85,B 0,C 180,E1 -9334.477,E2 -9334.477} C_VEL
LIN {X 0,Y 432.014,Z 307.49,A -85,B 0,C 180,E1 -9338.029,E2 -9338.029} C_VEL
LIN {X 0,Y 431.894,Z 313.437,A -85,B 0,C 180,E1 -9341.009,E2 -9341.009} C_VEL
LIN {X 0,Y 431.748,Z 319.371,A -85,B 0,C 180,E1 -9343.937,E2 -9343.937} C_VEL
LIN {X 0,Y 431.647,Z 327.28,A -85,B 0,C 180,E1 -9347.782,E2 -9347.782} C_VEL
LIN {X 0,Y 431.515,Z 331.996,A -85,B 0,C 180,E1 -9350.036,E2 -9350.036} C_VEL
LIN {X 0,Y 433.16,Z 343.673,A -85,B 0,C 180,E1 -9350.664,E2 -9350.664} C_VEL
LIN {X 0,Y 432.92,Z 353.668,A -85,B 0,C 180,E1 -9351.365,E2 -9351.365} C_VEL
LIN {X 0,Y 432.704,Z 361.838,A -85,B 0,C 180,E1 -9352.113,E2 -9352.113} C_VEL
LIN {X 0,Y 432.365,Z 369.859,A -85,B 0,C 180,E1 -9353.049,E2 -9353.049} C_VEL
LIN {X 0,Y 432.249,Z 377.243,A -85,B 0,C 180,E1 -9354.169,E2 -9354.169} C_VEL
LIN {X 0,Y 432.034,Z 383.133,A -85,B 0,C 180,E1 -9355.336,E2 -9355.336} C_VEL
LIN {X 0,Y 431.809,Z 388.255,A -85,B 0,C 180,E1 -9356.736,E2 -9356.736} C_VEL
LIN {X 0,Y 431.494,Z 391.622,A -85,B 0,C 180,E1 -9358.134,E2 -9358.134} C_VEL
LIN {X 0,Y 431.448,Z 392.967,A -85,B 0,C 180,E1 -9359.068,E2 -9359.068} C_VEL
LIN {X 0,Y 431.464,Z 393.629,A -85,B 0,C 180,E1 -9360.001,E2 -9360.001} C_VEL
LIN {X 0,Y 431.499,Z 393.625,A -85,B 0,C 180,E1 -9360.934,E2 -9360.934} C_VEL
LIN {X 0,Y 431.568,Z 392.956,A -85,B 0,C 180,E1 -9361.868,E2 -9361.868} C_VEL
LIN {X 0,Y 431.701,Z 391.611,A -85,B 0,C 180,E1 -9362.801,E2 -9362.801} C_VEL
LIN {X 0,Y 431.954,Z 389.553,A -85,B 0,C 180,E1 -9363.733,E2 -9363.733} C_VEL
LIN {X 0,Y 432.2,Z 386.749,A -85,B 0,C 180,E1 -9364.665,E2 -9364.665} C_VEL
LIN {X 0,Y 432.572,Z 382.052,A -85,B 0,C 180,E1 -9365.829,E2 -9365.829} C_VEL
LIN {X 0,Y 432.923,Z 375.822,A -85,B 0,C 180,E1 -9366.994,E2 -9366.994} C_VEL
LIN {X 0,Y 433.31,Z 368.926,A -85,B 0,C 180,E1 -9367.99,E2 -9367.99} C_VEL
LIN {X 0,Y 433.877,Z 360.144,A -85,B 0,C 180,E1 -9368.97,E2 -9368.97} C_VEL
LIN {X 0,Y 434.308,Z 350.704,A -85,B 0,C 180,E1 -9369.784,E2 -9369.784} C_VEL
LIN {X 0,Y 434.194,Z 345.77,A -85,B 0,C 180,E1 -9370.139,E2 -9370.139} C_VEL
LIN {X 0,Y 432.234,Z 336.171,A -85,B 0,C 180,E1 -9370.778,E2 -9370.778} C_VEL
LIN {X 0,Y 431.964,Z 334.859,A -85,B 0,C 180,E1 -9370.874,E2 -9370.874} C_VEL
LIN {X 0,Y 432.155,Z 330.466,A -85,B 0,C 180,E1 -9373.161,E2 -9373.161} C_VEL
LIN {X 0,Y 432.421,Z 324.244,A -85,B 0,C 180,E1 -9376.481,E2 -9376.481} C_VEL
LIN {X 0,Y 432.705,Z 317.975,A -85,B 0,C 180,E1 -9379.944,E2 -9379.944} C_VEL
LIN {X 0,Y 432.995,Z 312.788,A -85,B 0,C 180,E1 -9382.927,E2 -9382.927} C_VEL
LIN {X 0,Y 433.404,Z 307.703,A -85,B 0,C 180,E1 -9385.966,E2 -9385.966} C_VEL
LIN {X 0,Y 433.867,Z 302.726,A -85,B 0,C 180,E1 -9389.076,E2 -9389.076} C_VEL
LIN {X 0,Y 433.871,Z 299.632,A -85,B 0,C 180,E1 -9391.223,E2 -9391.223} C_VEL
LIN {X 0,Y 433.552,Z 296.774,A -85,B 0,C 180,E1 -9393.447,E2 -9393.447} C_VEL
LIN {X 0,Y 433.087,Z 294.211,A -85,B 0,C 180,E1 -9395.768,E2 -9395.768} C_VEL
LIN {X 0,Y 432.678,Z 292.117,A -85,B 0,C 180,E1 -9398.116,E2 -9398.116} C_VEL
LIN {X 0,Y 432.329,Z 290.634,A -85,B 0,C 180,E1 -9400.561,E2 -9400.561} C_VEL
LIN {X 0,Y 432.322,Z 290.635,A -85,B 0,C 180,E1 -9403.061,E2 -9403.061} C_VEL
LIN {X 0,Y 432.338,Z 290.633,A -85,B 0,C 180,E1 -9405.665,E2 -9405.665} C_VEL
LIN {X 0,Y 432.353,Z 290.765,A -85,B 0,C 180,E1 -9407.299,E2 -9407.299} C_VEL
LIN {X 0,Y 432.87,Z 292.723,A -85,B 0,C 180,E1 -9409.738,E2 -9409.738} C_VEL
LIN {X 0,Y 433.537,Z 295.512,A -85,B 0,C 180,E1 -9411.974,E2 -9411.974} C_VEL
LIN {X 0,Y 434.549,Z 299.497,A -85,B 0,C 180,E1 -9414.392,E2 -9414.392} C_VEL
LIN {X 0,Y 435.862,Z 304.969,A -85,B 0,C 180,E1 -9416.98,E2 -9416.98} C_VEL
LIN {X 0,Y 437.212,Z 311.715,A -85,B 0,C 180,E1 -9419.579,E2 -9419.579} C_VEL
LIN {X 0,Y 437.574,Z 315.035,A -85,B 0,C 180,E1 -9420.684,E2 -9420.684} C_VEL
LIN {X 0,Y 436.196,Z 323.796,A -85,B 0,C 180,E1 -9423.183,E2 -9423.183} C_VEL
LIN {X 0,Y 434.753,Z 335.184,A -85,B 0,C 180,E1 -9426.163,E2 -9426.163} C_VEL
LIN {X 0,Y 433.787,Z 346.146,A -85,B 0,C 180,E1 -9428.87,E2 -9428.87} C_VEL
LIN {X 0,Y 432.864,Z 359.69,A -85,B 0,C 180,E1 -9432.032,E2 -9432.032} C_VEL
LIN {X 0,Y 432.496,Z 367.007,A -85,B 0,C 180,E1 -9433.688,E2 -9433.688} C_VEL
LIN {X 0,Y 434.109,Z 380.324,A -85,B 0,C 180,E1 -9434.145,E2 -9434.145} C_VEL
LIN {X 0,Y 434.712,Z 392.868,A -85,B 0,C 180,E1 -9434.709,E2 -9434.709} C_VEL
LIN {X 0,Y 434.212,Z 404.134,A -85,B 0,C 180,E1 -9435.351,E2 -9435.351} C_VEL
LIN {X 0,Y 433.546,Z 415.264,A -85,B 0,C 180,E1 -9436.166,E2 -9436.166} C_VEL
LIN {X 0,Y 433.057,Z 426.659,A -85,B 0,C 180,E1 -9437.225,E2 -9437.225} C_VEL
LIN {X 0,Y 432.423,Z 435.816,A -85,B 0,C 180,E1 -9438.278,E2 -9438.278} C_VEL
LIN {X 0,Y 432.02,Z 444.232,A -85,B 0,C 180,E1 -9439.455,E2 -9439.455} C_VEL
LIN {X 0,Y 431.718,Z 452.477,A -85,B 0,C 180,E1 -9440.867,E2 -9440.867} C_VEL
LIN {X 0,Y 431.551,Z 458.055,A -85,B 0,C 180,E1 -9442.043,E2 -9442.043} C_VEL
LIN {X 0,Y 431.462,Z 463.773,A -85,B 0,C 180,E1 -9443.528,E2 -9443.528} C_VEL
LIN {X 0,Y 431.406,Z 467.737,A -85,B 0,C 180,E1 -9444.859,E2 -9444.859} C_VEL
LIN {X 0,Y 431.475,Z 470.86,A -85,B 0,C 180,E1 -9446.264,E2 -9446.264} C_VEL
LIN {X 0,Y 431.51,Z 472.347,A -85,B 0,C 180,E1 -9447.199,E2 -9447.199} C_VEL
LIN {X 0,Y 431.432,Z 473.4,A -85,B 0,C 180,E1 -9448.133,E2 -9448.133} C_VEL
LIN {X 0,Y 431.359,Z 474.046,A -85,B 0,C 180,E1 -9449.066,E2 -9449.066} C_VEL
LIN {X 0,Y 431.354,Z 474.244,A -85,B 0,C 180,E1 -9450,E2 -9450} C_VEL
LIN {X 0,Y 431.356,Z 474.012,A -85,B 0,C 180,E1 -9450.934,E2 -9450.934} C_VEL
LIN {X 0,Y 431.43,Z 473.38,A -85,B 0,C 180,E1 -9451.867,E2 -9451.867} C_VEL
LIN {X 0,Y 431.552,Z 472.318,A -85,B 0,C 180,E1 -9452.8,E2 -9452.8} C_VEL
LIN {X 0,Y 431.475,Z 470.762,A -85,B 0,C 180,E1 -9453.736,E2 -9453.736} C_VEL
LIN {X 0,Y 431.405,Z 467.583,A -85,B 0,C 180,E1 -9455.141,E2 -9455.141} C_VEL
LIN {X 0,Y 431.485,Z 463.281,A -85,B 0,C 180,E1 -9456.547,E2 -9456.547} C_VEL
LIN {X 0,Y 431.563,Z 457.711,A -85,B 0,C 180,E1 -9457.957,E2 -9457.957} C_VEL
LIN {X 0,Y 431.752,Z 450.682,A -85,B 0,C 180,E1 -9459.368,E2 -9459.368} C_VEL
LIN {X 0,Y 432.122,Z 441.795,A -85,B 0,C 180,E1 -9460.78,E2 -9460.78} C_VEL
LIN {X 0,Y 432.472,Z 432.629,A -85,B 0,C 180,E1 -9461.958,E2 -9461.958} C_VEL
LIN {X 0,Y 433.026,Z 424.542,A -85,B 0,C 180,E1 -9462.811,E2 -9462.811} C_VEL
LIN {X 0,Y 433.411,Z 414.632,A -85,B 0,C 180,E1 -9463.683,E2 -9463.683} C_VEL
LIN {X 0,Y 433.832,Z 404.114,A -85,B 0,C 180,E1 -9464.423,E2 -9464.423} C_VEL
LIN {X 0,Y 434.331,Z 392.193,A -85,B 0,C 180,E1 -9465.065,E2 -9465.065} C_VEL
LIN {X 0,Y 433.954,Z 384.684,A -85,B 0,C 180,E1 -9465.394,E2 -9465.394} C_VEL
LIN {X 0,Y 432.741,Z 372.165,A -85,B 0,C 180,E1 -9465.804,E2 -9465.804} C_VEL
LIN {X 0,Y 432.352,Z 368.07,A -85,B 0,C 180,E1 -9465.921,E2 -9465.921} C_VEL
LIN {X 0,Y 433.055,Z 354.611,A -85,B 0,C 180,E1 -9468.94,E2 -9468.94} C_VEL
LIN {X 0,Y 434.007,Z 339.993,A -85,B 0,C 180,E1 -9472.268,E2 -9472.268} C_VEL
LIN {X 0,Y 435.217,Z 324.558,A -85,B 0,C 180,E1 -9475.849,E2 -9475.849} C_VEL
LIN {X 0,Y 436.416,Z 311.712,A -85,B 0,C 180,E1 -9478.889,E2 -9478.889} C_VEL
LIN {X 0,Y 435.909,Z 307.381,A -85,B 0,C 180,E1 -9479.987,E2 -9479.987} C_VEL
LIN {X 0,Y 433.534,Z 296.24,A -85,B 0,C 180,E1 -9482.968,E2 -9482.968} C_VEL
LIN {X 0,Y 432.383,Z 290.629,A -85,B 0,C 180,E1 -9484.538,E2 -9484.538} C_VEL
LIN {X 0,Y 432.342,Z 290.633,A -85,B 0,C 180,E1 -9488.15,E2 -9488.15} C_VEL
LIN {X 0,Y 432.338,Z 290.632,A -85,B 0,C 180,E1 -9491.602,E2 -9491.602} C_VEL
LIN {X 0,Y 432.339,Z 290.633,A -85,B 0,C 180,E1 -9494.347,E2 -9494.347} C_VEL
LIN {X 0,Y 432.326,Z 290.633,A -85,B 0,C 180,E1 -9497.015,E2 -9497.015} C_VEL
LIN {X 0,Y 432.342,Z 290.631,A -85,B 0,C 180,E1 -9499.82,E2 -9499.82} C_VEL
LIN {X 0,Y 432.312,Z 290.636,A -85,B 0,C 180,E1 -9503.021,E2 -9503.021} C_VEL
LIN {X 0,Y 432.363,Z 290.632,A -85,B 0,C 180,E1 -9505.996,E2 -9505.996} C_VEL
LIN {X 0,Y 432.33,Z 290.637,A -85,B 0,C 180,E1 -9509.494,E2 -9509.494} C_VEL
LIN {X 0,Y 432.312,Z 290.694,A -85,B 0,C 180,E1 -9510.274,E2 -9510.274} C_VEL
LIN {X 0,Y 432.694,Z 293.321,A -85,B 0,C 180,E1 -9511.294,E2 -9511.294} C_VEL
LIN {X 0,Y 432.581,Z 301.651,A -85,B 0,C 180,E1 -9514.497,E2 -9514.497} C_VEL
LIN {X 0,Y 432.497,Z 307.958,A -85,B 0,C 180,E1 -9517.045,E2 -9517.045} C_VEL
LIN {X 0,Y 432.475,Z 315.328,A -85,B 0,C 180,E1 -9520.045,E2 -9520.045} C_VEL
LIN {X 0,Y 432.367,Z 323.632,A -85,B 0,C 180,E1 -9523.543,E2 -9523.543} C_VEL
LIN {X 0,Y 432.305,Z 331.314,A -85,B 0,C 180,E1 -9526.843,E2 -9526.843} C_VEL
LIN {X 0,Y 432.254,Z 336.805,A -85,B 0,C 180,E1 -9529.222,E2 -9529.222} C_VEL
LIN {X 0,Y 432.29,Z 338.914,A -85,B 0,C 180,E1 -9530.141,E2 -9530.141} C_VEL
LIN {X 0,Y 433.592,Z 346.39,A -85,B 0,C 180,E1 -9530.553,E2 -9530.553} C_VEL
LIN {X 0,Y 433.355,Z 355.35,A -85,B 0,C 180,E1 -9531.136,E2 -9531.136} C_VEL
LIN {X 0,Y 433.075,Z 364.307,A -85,B 0,C 180,E1 -9531.93,E2 -9531.93} C_VEL
LIN {X 0,Y 432.753,Z 369.692,A -85,B 0,C 180,E1 -9532.534,E2 -9532.534} C_VEL
LIN {X 0,Y 432.593,Z 376.366,A -85,B 0,C 180,E1 -9533.469,E2 -9533.469} C_VEL
LIN {X 0,Y 432.338,Z 381.492,A -85,B 0,C 180,E1 -9534.402,E2 -9534.402} C_VEL
LIN {X 0,Y 432.184,Z 385.517,A -85,B 0,C 180,E1 -9535.335,E2 -9535.335} C_VEL
LIN {X 0,Y 431.947,Z 388.645,A -85,B 0,C 180,E1 -9536.267,E2 -9536.267} C_VEL
LIN {X 0,Y 431.672,Z 390.961,A -85,B 0,C 180,E1 -9537.199,E2 -9537.199} C_VEL
LIN {X 0,Y 431.541,Z 392.5,A -85,B 0,C 180,E1 -9538.132,E2 -9538.132} C_VEL
LIN {X 0,Y 431.476,Z 393.321,A -85,B 0,C 180,E1 -9539.066,E2 -9539.066} C_VEL
LIN {X 0,Y 431.44,Z 393.452,A -85,B 0,C 180,E1 -9539.999,E2 -9539.999} C_VEL
